KUKA KRL program: MyProgram_140().src

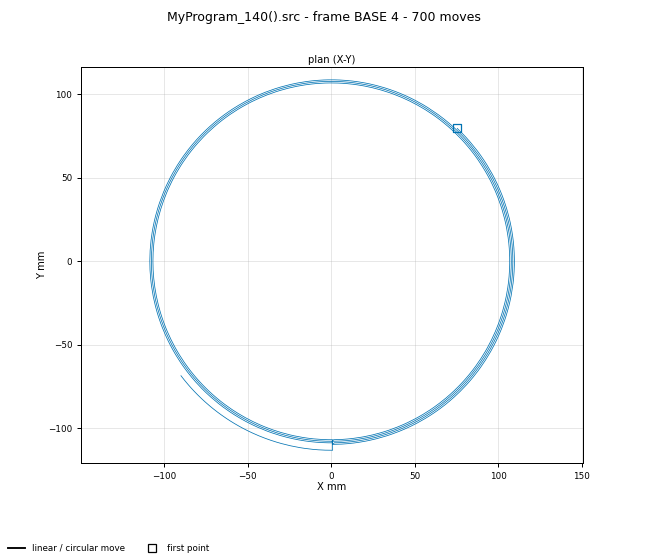
[picture p0: tool path of MyProgram_140().src in frame BASE 4, 700 of 700 moves have a stored position in this frame; points joined in program order, loops and branches not executed]
&ACCESS RVP
&REL 1
&PARAM TEMPLATE = C:\KRC\Roboter\Template\vorgabe
&PARAM EDITMASK = *
DEF MyProgram_140()
; ---- Setting reference (Base) ----
$BASE = BASE_DATA[4]

; --------------------------
; ---- Setting tool (TCP) ----
$TOOL = TOOL_DATA[3]
; --------------------------

$VEL.CP = VEL_APROX_PRINT
Startdeposition()
$VEL.CP = VEL_PRINT
LIN {X 75.377,Y 79.5533,Z 112,A 41.5429,B 24.9329,C -1.8914,E1 25.1111,E2 404.2043} C_DIS
LIN {X 77.9618,Y 77.0209,Z 112,A 39.7564,B 24.9329,C -1.8919,E1 25.1146,E2 405.9821} C_DIS
LIN {X 80.4801,Y 74.3866,Z 112,A 37.7745,B 24.9334,C -1.8843,E1 25.1184,E2 407.9731} C_DIS
LIN {X 82.9193,Y 71.6588,Z 112,A 35.8331,B 24.9338,C -1.8787,E1 25.122,E2 409.9192} C_DIS
LIN {X 87.2481,Y 66.3205,Z 112,A 32.4353,B 24.9338,C -1.8785,E1 25.1279,E2 413.3016} C_DIS
LIN {X 89.2094,Y 63.6549,Z 112,A 30.167,B 24.9358,C -1.8509,E1 25.1317,E2 415.624} C_DIS
LIN {X 91.3083,Y 60.6066,Z 112,A 28.6448,B 24.9349,C -1.8637,E1 25.134,E2 417.1083} C_DIS
LIN {X 93.1243,Y 57.7775,Z 112,A 27.0143,B 24.9349,C -1.8646,E1 25.1364,E2 418.7285} C_DIS
LIN {X 96.3793,Y 52.1661,Z 112,A 23.6682,B 24.9353,C -1.8574,E1 25.1411,E2 422.0744} C_DIS
LIN {X 97.758,Y 49.5356,Z 112,A 21.4703,B 24.9376,C -1.825,E1 25.1439,E2 424.3371} C_DIS
LIN {X 99.5673,Y 45.7914,Z 112,A 20.1073,B 24.9356,C -1.8541,E1 25.1455,E2 425.6239} C_DIS
LIN {X 101.01,Y 42.5115,Z 112,A 18.0918,B 24.9364,C -1.8425,E1 25.1477,E2 427.6559} C_DIS
LIN {X 102.2498,Y 39.4421,Z 112,A 15.9159,B 24.9381,C -1.8179,E1 25.15,E2 429.8778} C_DIS
LIN {X 103.3582,Y 36.433,Z 112,A 14.9671,B 24.9362,C -1.8448,E1 25.1508,E2 430.7576} C_DIS
LIN {X 104.9128,Y 31.6824,Z 112,A 11.8359,B 24.9383,C -1.8141,E1 25.1535,E2 433.9435} C_DIS
LIN {X 106.5712,Y 25.5542,Z 112,A 8.8976,B 24.9379,C -1.8206,E1 25.1556,E2 436.8496} C_DIS
LIN {X 107.1441,Y 23.0328,Z 112,A 7.4205,B 24.9385,C -1.8109,E1 25.1565,E2 438.341} C_DIS
LIN {X 107.8727,Y 19.3326,Z 112,A 5.4382,B 24.939,C -1.8042,E1 25.1575,E2 440.3275} C_DIS
LIN {X 108.4862,Y 15.5247,Z 112,A 3.44,B 24.9394,C -1.7986,E1 25.1583,E2 442.3271} C_DIS
LIN {X 108.9203,Y 12.1254,Z 112,A 1.543,B 24.9401,C -1.7882,E1 25.159,E2 444.2375} C_DIS
LIN {X 109.2712,Y 8.3779,Z 112,A -0.353,B 24.9403,C -1.7851,E1 25.1594,E2 446.1296} C_DIS
LIN {X 109.4863,Y 4.7961,Z 112,A -2.1281,B 24.9403,C -1.7835,E1 25.1597,E2 447.8979} C_DIS
LIN {X 109.5863,Y 1.1777,Z 112,A -4.0411,B 24.9409,C -1.7764,E1 25.1597,E2 449.8161} C_DIS
LIN {X 109.5675,Y -2.3032,Z 112,A -5.9034,B 24.9414,C -1.7686,E1 25.1597,E2 451.6858} C_DIS
LIN {X 109.4279,Y -5.9824,Z 112,A -7.7314,B 24.9415,C -1.7667,E1 25.1595,E2 453.5075} C_DIS
LIN {X 109.1646,Y -9.6696,Z 112,A -9.7033,B 24.942,C -1.7587,E1 25.159,E2 455.4866} C_DIS
LIN {X 108.816,Y -13.0152,Z 112,A -11.5187,B 24.9426,C -1.7504,E1 25.1585,E2 457.3107} C_DIS
LIN {X 107.6217,Y -20.684,Z 112,A -15.0658,B 24.9419,C -1.76,E1 25.1569,E2 460.8144} C_DIS
LIN {X 106.7931,Y -24.6068,Z 112,A -17.514,B 24.9434,C -1.7375,E1 25.1555,E2 463.3013} C_DIS
LIN {X 105.883,Y -28.2691,Z 112,A -19.5465,B 24.944,C -1.7286,E1 25.154,E2 465.3432} C_DIS
LIN {X 104.8011,Y -32.0495,Z 112,A -21.5394,B 24.9442,C -1.7248,E1 25.1525,E2 467.3336} C_DIS
LIN {X 103.8,Y -35.1546,Z 112,A -23.2039,B 24.9445,C -1.7213,E1 25.151,E2 468.9969} C_DIS
LIN {X 101.7907,Y -40.6108,Z 112,A -26.0892,B 24.9446,C -1.7186,E1 25.1482,E2 471.8725} C_DIS
LIN {X 100.2347,Y -44.3123,Z 112,A -28.8953,B 24.947,C -1.681,E1 25.145,E2 474.7519} C_DIS
LIN {X 98.5105,Y -48.0243,Z 112,A -30.3569,B 24.9456,C -1.7044,E1 25.1433,E2 476.1506} C_DIS
LIN {X 97.1937,Y -50.6336,Z 112,A -32.1386,B 24.9466,C -1.6886,E1 25.141,E2 477.96} C_DIS
LIN {X 95.3849,Y -53.9661,Z 112,A -34.0746,B 24.9468,C -1.6848,E1 25.1384,E2 479.8949} C_DIS
LIN {X 92.3521,Y -59.0034,Z 112,A -36.8045,B 24.9464,C -1.6912,E1 25.1345,E2 482.5959} C_DIS
LIN {X 89.3255,Y -63.492,Z 112,A -39.5066,B 24.9466,C -1.6888,E1 25.1303,E2 485.2901} C_DIS
LIN {X 87.7889,Y -65.6007,Z 112,A -41.8928,B 24.9496,C -1.6403,E1 25.1261,E2 487.7794} C_DIS
LIN {X 84.8508,Y -69.36,Z 112,A -44.0527,B 24.9491,C -1.6482,E1 25.1223,E2 489.9107} C_DIS
LIN {X 82.6946,Y -71.9159,Z 112,A -45.1241,B 24.9475,C -1.6733,E1 25.1205,E2 490.9181} C_DIS
LIN {X 80.8114,Y -74.0256,Z 112,A -46.889,B 24.9486,C -1.6569,E1 25.1171,E2 492.7137} C_DIS
LIN {X 77.0376,Y -77.9452,Z 112,A -50.0153,B 24.9498,C -1.6376,E1 25.1109,E2 495.8723} C_DIS
LIN {X 73.6027,Y -81.1994,Z 112,A -52.2586,B 24.9495,C -1.6417,E1 25.1064,E2 498.0968} C_DIS
LIN {X 70.6465,Y -83.7833,Z 112,A -54.5965,B 24.9505,C -1.6247,E1 25.1014,E2 500.4658} C_DIS
LIN {X 68.0835,Y -85.8773,Z 112,A -56.4348,B 24.9511,C -1.6162,E1 25.0973,E2 502.3171} C_DIS
LIN {X 64.9846,Y -88.246,Z 112,A -57.6863,B 24.9492,C -1.646,E1 25.0947,E2 503.4939} C_DIS
LIN {X 61.6206,Y -90.6267,Z 112,A -60.4571,B 24.9511,C -1.6149,E1 25.0882,E2 506.3286} C_DIS
LIN {X 58.8929,Y -92.423,Z 112,A -61.4446,B 24.9494,C -1.6427,E1 25.086,E2 507.2473} C_DIS
LIN {X 56.1138,Y -94.1364,Z 112,A -63.2822,B 24.95,C -1.6337,E1 25.0816,E2 509.1002} C_DIS
LIN {X 51.5128,Y -96.7304,Z 112,A -66.8077,B 24.9523,C -1.5961,E1 25.0728,E2 512.7044} C_DIS
LIN {X 47.8579,Y -98.5904,Z 112,A -68.1842,B 24.9505,C -1.6253,E1 25.0695,E2 514.0081} C_DIS
LIN {X 43.812,Y -100.4528,Z 112,A -70.6813,B 24.9512,C -1.6145,E1 25.0631,E2 516.5246} C_DIS
LIN {X 40.4857,Y -101.8399,Z 112,A -73.4033,B 24.9534,C -1.5763,E1 25.0559,E2 519.3307} C_DIS
LIN {X 35.6056,Y -103.6479,Z 112,A -75.1848,B 24.9513,C -1.6124,E1 25.0514,E2 521.0232} C_DIS
LIN {X 32.8161,Y -104.5634,Z 112,A -77.2633,B 24.9528,C -1.5876,E1 25.0457,E2 523.1566} C_DIS
LIN {X 29.377,Y -105.5818,Z 112,A -78.6243,B 24.9516,C -1.6072,E1 25.0422,E2 524.4689} C_DIS
LIN {X 27.077,Y -106.1938,Z 112,A -80.5198,B 24.9533,C -1.5786,E1 25.0369,E2 526.4294} C_DIS
LIN {X 23.0114,Y -107.1488,Z 112,A -81.9602,B 24.9516,C -1.6077,E1 25.0332,E2 527.7989} C_DIS
LIN {X 20.5758,Y -107.6425,Z 112,A -83.3737,B 24.9519,C -1.6018,E1 25.0292,E2 529.2248} C_DIS
LIN {X 16.5964,Y -108.3275,Z 112,A -85.5038,B 24.9521,C -1.5994,E1 25.0234,E2 531.3583} C_DIS
LIN {X 13.46,Y -108.7634,Z 112,A -87.2798,B 24.9524,C -1.5932,E1 25.0184,E2 533.1475} C_DIS
LIN {X 9.8662,Y -109.1465,Z 112,A -89.0287,B 24.9521,C -1.5981,E1 25.0136,E2 534.8837} C_DIS
LIN {X 6.2606,Y -109.4125,Z 112,A -90.9395,B 24.9522,C -1.5964,E1 25.0082,E2 536.7978} C_DIS
LIN {X 2.6896,Y -109.5604,Z 112,A -92.7328,B 24.9522,C -1.5988,E1 25.0033,E2 538.5848} C_DIS
LIN {X 0.7741,Y -109.5863,Z 112,A -93.6774,B 24.952,C -1.601,E1 25.0006,E2 539.5242} C_DIS
Enddeposition()
LIN {X 0.7741,Y -109.5863,Z 112,A -93.6774,B 24.952,C -1.601,E1 25.0006,E2 539.5242} C_DIS
Startdeposition()
$VEL.CP = VEL_PRINT
LIN {X 1.7946,Y -108.6458,Z 112,A -92.6033,B 24.9496,C -1.6396,E1 25.0039,E2 538.3587} C_DIS
LIN {X 4.823,Y -108.5535,Z 112,A -90.9393,B 24.9494,C -1.643,E1 25.0086,E2 536.6872} C_DIS
LIN {X 8.3887,Y -108.3365,Z 112,A -89.0175,B 24.9493,C -1.6454,E1 25.0139,E2 534.7604} C_DIS
LIN {X 11.9173,Y -108.0066,Z 112,A -87.0722,B 24.949,C -1.6497,E1 25.0193,E2 532.8063} C_DIS
LIN {X 15.0872,Y -107.6081,Z 112,A -85.4658,B 24.9491,C -1.6475,E1 25.0238,E2 531.2064} C_DIS
LIN {X 18.76,Y -107.0298,Z 112,A -83.4639,B 24.9489,C -1.6507,E1 25.0293,E2 529.1988} C_DIS
LIN {X 22.7045,Y -106.2629,Z 112,A -80.8395,B 24.9475,C -1.6741,E1 25.0366,E2 526.5224} C_DIS
LIN {X 26.6242,Y -105.349,Z 112,A -79.2573,B 24.9488,C -1.6532,E1 25.0408,E2 524.992} C_DIS
LIN {X 32.0291,Y -103.8328,Z 112,A -76.2746,B 24.9485,C -1.6575,E1 25.0488,E2 522.0042} C_DIS
LIN {X 35.4323,Y -102.7228,Z 112,A -74.419,B 24.9485,C -1.6585,E1 25.0537,E2 520.15} C_DIS
LIN {X 40.5582,Y -100.8083,Z 112,A -71.5163,B 24.9482,C -1.6632,E1 25.0613,E2 517.2424} C_DIS
LIN {X 43.2349,Y -99.6889,Z 112,A -69.482,B 24.9466,C -1.6873,E1 25.0666,E2 515.156} C_DIS
LIN {X 46.9131,Y -98.0116,Z 112,A -68.0486,B 24.9483,C -1.6605,E1 25.0701,E2 513.7897} C_DIS
LIN {X 48.9246,Y -97.0243,Z 112,A -66.0205,B 24.9459,C -1.6992,E1 25.0753,E2 511.6757} C_DIS
LIN {X 53.0461,Y -94.8325,Z 112,A -64.3618,B 24.9478,C -1.6686,E1 25.0792,E2 510.0941} C_DIS
LIN {X 56.0148,Y -93.1111,Z 112,A -62.5662,B 24.9477,C -1.6713,E1 25.0835,E2 508.2976} C_DIS
LIN {X 59.0835,Y -91.1945,Z 112,A -60.1603,B 24.9461,C -1.6967,E1 25.0893,E2 505.8395} C_DIS
LIN {X 61.9282,Y -89.2861,Z 112,A -58.7501,B 24.9469,C -1.6831,E1 25.0925,E2 504.4662} C_DIS
LIN {X 65.7981,Y -86.4746,Z 112,A -56.1025,B 24.9462,C -1.6939,E1 25.0984,E2 501.8027} C_DIS
LIN {X 70.9814,Y -82.2747,Z 112,A -52.6965,B 24.946,C -1.6968,E1 25.1057,E2 498.4027} C_DIS
LIN {X 73.5373,Y -79.996,Z 112,A -50.3929,B 24.9444,C -1.7231,E1 25.1106,E2 496.0464} C_DIS
LIN {X 76.5543,Y -77.1142,Z 112,A -48.1485,B 24.9439,C -1.7305,E1 25.115,E2 493.7941} C_DIS
LIN {X 79.6532,Y -73.911,Z 112,A -46.3962,B 24.9452,C -1.7099,E1 25.1183,E2 492.0981} C_DIS
LIN {X 81.5881,Y -71.7678,Z 112,A -44.2717,B 24.9432,C -1.7405,E1 25.1223,E2 489.9107} C_DIS
LIN {X 84.4673,Y -68.3547,Z 112,A -42.3211,B 24.944,C -1.7288,E1 25.1257,E2 487.9969} C_DIS
LIN {X 88.438,Y -63.1333,Z 112,A -38.1967,B 24.9414,C -1.7681,E1 25.1326,E2 483.7997} C_DIS
LIN {X 91.6609,Y -58.3569,Z 112,A -35.9253,B 24.9431,C -1.7424,E1 25.1359,E2 481.6004} C_DIS
LIN {X 93.7475,Y -54.9424,Z 112,A -34.0234,B 24.9433,C -1.7392,E1 25.1386,E2 479.7157} C_DIS
LIN {X 95.2658,Y -52.2666,Z 112,A -32.5867,B 24.9435,C -1.7358,E1 25.1406,E2 478.2946} C_DIS
LIN {X 97.5098,Y -47.9483,Z 112,A -29.1045,B 24.9403,C -1.7844,E1 25.1451,E2 474.7162} C_DIS
LIN {X 99.5831,Y -43.4777,Z 112,A -27.3196,B 24.9422,C -1.7559,E1 25.147,E2 473.0083} C_DIS
LIN {X 100.6196,Y -41.0219,Z 112,A -25.5416,B 24.9408,C -1.7769,E1 25.1489,E2 471.1906} C_DIS
LIN {X 101.8245,Y -37.9368,Z 112,A -24.2243,B 24.9417,C -1.7631,E1 25.1502,E2 469.9131} C_DIS
LIN {X 102.8382,Y -35.0935,Z 112,A -22.5787,B 24.9412,C -1.7705,E1 25.1517,E2 468.2593} C_DIS
LIN {X 103.8368,Y -32.0163,Z 112,A -20.9416,B 24.9411,C -1.7728,E1 25.1531,E2 466.626} C_DIS
LIN {X 104.7149,Y -29.0219,Z 112,A -19.1378,B 24.9403,C -1.7851,E1 25.1544,E2 464.8035} C_DIS
LIN {X 105.6382,Y -25.4512,Z 112,A -17.2444,B 24.94,C -1.7891,E1 25.1557,E2 462.9118} C_DIS
LIN {X 106.4295,Y -21.9056,Z 112,A -15.1285,B 24.939,C -1.8042,E1 25.157,E2 460.7725} C_DIS
LIN {X 107.4359,Y -16.2708,Z 112,A -12.2941,B 24.9389,C -1.8057,E1 25.1582,E2 457.9511} C_DIS
LIN {X 107.9465,Y -12.4376,Z 112,A -10.3554,B 24.9387,C -1.8079,E1 25.1589,E2 456.0188} C_DIS
LIN {X 108.3235,Y -8.5506,Z 112,A -8.3385,B 24.9384,C -1.8127,E1 25.1594,E2 454.0025} C_DIS
LIN {X 108.5553,Y -4.7801,Z 112,A -6.3472,B 24.938,C -1.8191,E1 25.1597,E2 452.0079} C_DIS
LIN {X 108.6585,Y -0.7391,Z 112,A -4.2535,B 24.9376,C -1.8244,E1 25.1597,E2 449.9143} C_DIS
LIN {X 108.6205,Y 2.9676,Z 112,A -2.291,B 24.9372,C -1.831,E1 25.1597,E2 447.9477} C_DIS
LIN {X 108.4705,Y 6.4379,Z 112,A -0.4958,B 24.9369,C -1.8353,E1 25.1594,E2 446.1531} C_DIS
LIN {X 108.2062,Y 9.925,Z 112,A 1.3366,B 24.9365,C -1.8408,E1 25.159,E2 444.3188} C_DIS
LIN {X 107.7971,Y 13.6733,Z 112,A 3.2648,B 24.9362,C -1.8444,E1 25.1584,E2 442.3932} C_DIS
LIN {X 107.4067,Y 16.4592,Z 112,A 4.7603,B 24.9359,C -1.8497,E1 25.1578,E2 440.8942} C_DIS
LIN {X 106.8273,Y 19.8864,Z 112,A 6.707,B 24.9351,C -1.8605,E1 25.1568,E2 438.9333} C_DIS
LIN {X 106.1072,Y 23.4184,Z 112,A 8.4034,B 24.9353,C -1.8574,E1 25.1558,E2 437.2542} C_DIS
LIN {X 104.6842,Y 29.1302,Z 112,A 12.1394,B 24.9327,C -1.8951,E1 25.1531,E2 433.4508} C_DIS
LIN {X 103.5197,Y 33.0295,Z 112,A 13.8129,B 24.9337,C -1.8806,E1 25.1518,E2 431.821} C_DIS
LIN {X 102.3599,Y 36.4666,Z 112,A 15.4437,B 24.9342,C -1.8738,E1 25.1503,E2 430.2153} C_DIS
LIN {X 101.3028,Y 39.307,Z 112,A 17.1938,B 24.9334,C -1.8853,E1 25.1485,E2 428.448} C_DIS
LIN {X 100.0814,Y 42.3182,Z 112,A 18.9048,B 24.933,C -1.8902,E1 25.1467,E2 426.7348} C_DIS
LIN {X 98.6024,Y 45.6585,Z 112,A 21.3213,B 24.9311,C -1.9174,E1 25.1438,E2 424.2673} C_DIS
LIN {X 96.9145,Y 49.1405,Z 112,A 22.8666,B 24.9322,C -1.9012,E1 25.142,E2 422.7683} C_DIS
LIN {X 95.2954,Y 52.212,Z 112,A 25.2882,B 24.93,C -1.9323,E1 25.1386,E2 420.286} C_DIS
LIN {X 93.1242,Y 55.9932,Z 112,A 27.0114,B 24.9314,C -1.9131,E1 25.1363,E2 418.6171} C_DIS
LIN {X 91.2048,Y 59.0675,Z 112,A 28.8675,B 24.9312,C -1.9157,E1 25.1335,E2 416.7641} C_DIS
LIN {X 87.762,Y 64.0698,Z 112,A 31.9965,B 24.9308,C -1.9206,E1 25.1285,E2 413.6389} C_DIS
LIN {X 83.1642,Y 69.9372,Z 112,A 36.026,B 24.9299,C -1.9342,E1 25.1214,E2 409.5959} C_DIS
LIN {X 80.7592,Y 72.6989,Z 112,A 37.9225,B 24.9296,C -1.9372,E1 25.1179,E2 407.701} C_DIS
LIN {X 78.2275,Y 75.4158,Z 112,A 39.7969,B 24.9296,C -1.9379,E1 25.1143,E2 405.833} C_DIS
LIN {X 75.5755,Y 78.0736,Z 112,A 41.7857,B 24.9293,C -1.9425,E1 25.1104,E2 403.8417} C_DIS
LIN {X 72.9803,Y 80.5071,Z 112,A 43.7462,B 24.9287,C -1.95,E1 25.1063,E2 401.8715} C_DIS
LIN {X 70.3797,Y 82.7877,Z 112,A 45.4481,B 24.9288,C -1.9483,E1 25.1027,E2 400.1801} C_DIS
LIN {X 67.5295,Y 85.1287,Z 112,A 48.0314,B 24.9265,C -1.9795,E1 25.097,E2 397.5329} C_DIS
LIN {X 64.0831,Y 87.7523,Z 112,A 49.6382,B 24.9284,C -1.9544,E1 25.0935,E2 395.9912} C_DIS
LIN {X 57.7373,Y 92.0518,Z 112,A 53.6998,B 24.9278,C -1.9617,E1 25.0841,E2 391.9257} C_DIS
LIN {X 54.769,Y 93.8499,Z 112,A 55.4275,B 24.928,C -1.9601,E1 25.0799,E2 390.2073} C_DIS
LIN {X 49.9797,Y 96.4856,Z 112,A 58.3902,B 24.9274,C -1.9674,E1 25.0726,E2 387.2358} C_DIS
LIN {X 47.5326,Y 97.714,Z 112,A 60.3077,B 24.9258,C -1.9892,E1 25.0677,E2 385.2717} C_DIS
LIN {X 44.2589,Y 99.2392,Z 112,A 61.825,B 24.9269,C -1.9751,E1 25.0639,E2 383.7917} C_DIS
LIN {X 40.9639,Y 100.6432,Z 112,A 63.5708,B 24.9272,C -1.9711,E1 25.0595,E2 382.0593} C_DIS
LIN {X 38.3632,Y 101.663,Z 112,A 65.5197,B 24.9256,C -1.9925,E1 25.0543,E2 380.064} C_DIS
LIN {X 35.071,Y 102.8458,Z 112,A 66.9096,B 24.9269,C -1.975,E1 25.0507,E2 378.7182} C_DIS
LIN {X 31.9792,Y 103.8483,Z 112,A 68.6432,B 24.9267,C -1.9772,E1 25.0461,E2 376.9826} C_DIS
LIN {X 27.1829,Y 105.2055,Z 112,A 71.8741,B 24.9247,C -2.004,E1 25.0372,E2 373.6933} C_DIS
LIN {X 23.0994,Y 106.1768,Z 112,A 73.4715,B 24.9265,C -1.9796,E1 25.033,E2 372.156} C_DIS
LIN {X 20.474,Y 106.7142,Z 112,A 74.9013,B 24.9265,C -1.9809,E1 25.0291,E2 370.7248} C_DIS
LIN {X 16.3963,Y 107.4165,Z 112,A 77.1625,B 24.9261,C -1.9848,E1 25.0228,E2 368.4565} C_DIS
LIN {X 12.6448,Y 107.9222,Z 112,A 79.0915,B 24.9263,C -1.9825,E1 25.0175,E2 366.5344} C_DIS
LIN {X 8.7801,Y 108.3052,Z 112,A 81.1507,B 24.9263,C -1.9832,E1 25.0118,E2 364.4749} C_DIS
LIN {X 5.1053,Y 108.5413,Z 112,A 83.076,B 24.9263,C -1.9825,E1 25.0064,E2 362.552} C_DIS
LIN {X 2.0105,Y 108.6418,Z 112,A 84.7124,B 24.9263,C -1.9825,E1 25.0019,E2 360.916} C_DIS
LIN {X -1.8793,Y 108.6443,Z 112,A 86.6636,B 24.9266,C -1.9779,E1 24.9964,E2 358.9755} C_DIS
LIN {X -4.5203,Y 108.5665,Z 112,A 88.1228,B 24.9265,C -1.9802,E1 24.9924,E2 357.5107} C_DIS
LIN {X -8.1438,Y 108.3561,Z 112,A 90.1157,B 24.9263,C -1.9825,E1 24.9868,E2 355.5114} C_DIS
LIN {X -11.5164,Y 108.0486,Z 112,A 91.9035,B 24.9263,C -1.9817,E1 24.9818,E2 353.7246} C_DIS
LIN {X -15.1504,Y 107.5991,Z 112,A 93.6701,B 24.9269,C -1.974,E1 24.977,E2 351.9751} C_DIS
LIN {X -20.548,Y 106.6999,Z 112,A 97.2399,B 24.9251,C -1.9992,E1 24.967,E2 348.3418} C_DIS
LIN {X -24.5356,Y 105.8542,Z 112,A 98.7968,B 24.927,C -1.9735,E1 24.9629,E2 346.8438} C_DIS
LIN {X -30.2104,Y 104.3781,Z 112,A 102.4845,B 24.9255,C -1.994,E1 24.9528,E2 343.1018} C_DIS
LIN {X -34.0854,Y 103.1781,Z 112,A 104.1442,B 24.9271,C -1.9724,E1 24.9486,E2 341.4904} C_DIS
LIN {X -37.0469,Y 102.1502,Z 112,A 105.7169,B 24.9274,C -1.9672,E1 24.9444,E2 339.927} C_DIS
LIN {X -39.4458,Y 101.2483,Z 112,A 107.5174,B 24.9263,C -1.983,E1 24.9397,E2 338.0849} C_DIS
LIN {X -42.7406,Y 99.9027,Z 112,A 109.0294,B 24.9275,C -1.9659,E1 24.9359,E2 336.61} C_DIS
LIN {X -45.2802,Y 98.7785,Z 112,A 110.8572,B 24.9266,C -1.978,E1 24.9312,E2 334.7491} C_DIS
LIN {X -48.3038,Y 97.3336,Z 112,A 112.6602,B 24.9268,C -1.9765,E1 24.9266,E2 332.9447} C_DIS
LIN {X -51.5219,Y 95.6697,Z 112,A 114.406,B 24.9275,C -1.9668,E1 24.9224,E2 331.2171} C_DIS
LIN {X -55.5157,Y 93.4086,Z 112,A 116.6397,B 24.9283,C -1.9552,E1 24.917,E2 329.0044} C_DIS
LIN {X -59.0398,Y 91.2226,Z 112,A 118.6379,B 24.9292,C -1.9438,E1 24.9124,E2 327.0271} C_DIS
LIN {X -61.302,Y 89.7182,Z 112,A 120.6482,B 24.9277,C -1.9633,E1 24.9076,E2 324.9635} C_DIS
LIN {X -64.2075,Y 87.6612,Z 112,A 122.0568,B 24.9293,C -1.9413,E1 24.9045,E2 323.6024} C_DIS
LIN {X -67.0333,Y 85.5209,Z 112,A 123.7482,B 24.9301,C -1.9305,E1 24.9008,E2 321.9306} C_DIS
LIN {X -69.5994,Y 83.4449,Z 112,A 126.1945,B 24.9284,C -1.9538,E1 24.8954,E2 319.4194} C_DIS
LIN {X -72.4368,Y 80.9939,Z 112,A 127.6579,B 24.9302,C -1.9295,E1 24.8925,E2 318.0081} C_DIS
LIN {X -75.1131,Y 78.5193,Z 112,A 129.4026,B 24.931,C -1.9182,E1 24.889,E2 316.2833} C_DIS
LIN {X -78.1859,Y 75.459,Z 112,A 132.3647,B 24.9296,C -1.9384,E1 24.883,E2 313.2602} C_DIS
LIN {X -80.6542,Y 72.8162,Z 112,A 133.8743,B 24.931,C -1.9184,E1 24.8803,E2 311.7917} C_DIS
LIN {X -83.1284,Y 69.9798,Z 112,A 135.722,B 24.9318,C -1.908,E1 24.8769,E2 309.9603} C_DIS
LIN {X -85.5795,Y 66.9591,Z 112,A 138.1312,B 24.9312,C -1.9162,E1 24.8727,E2 307.5203} C_DIS
LIN {X -88.378,Y 63.2174,Z 112,A 140.3479,B 24.9323,C -1.9001,E1 24.8691,E2 305.3313} C_DIS
LIN {X -90.2079,Y 60.5789,Z 112,A 142.5634,B 24.9312,C -1.9152,E1 24.8656,E2 303.0687} C_DIS
LIN {X -92.2077,Y 57.4877,Z 112,A 144.9067,B 24.9305,C -1.9251,E1 24.8621,E2 300.69} C_DIS
LIN {X -94.9198,Y 52.8897,Z 112,A 146.7523,B 24.9337,C -1.88,E1 24.8597,E2 298.9423} C_DIS
LIN {X -96.5074,Y 49.937,Z 112,A 148.4926,B 24.9342,C -1.8737,E1 24.8574,E2 297.2076} C_DIS
LIN {X -98.8674,Y 45.0839,Z 112,A 151.562,B 24.9342,C -1.8735,E1 24.8537,E2 294.122} C_DIS
LIN {X -100.4255,Y 41.4987,Z 112,A 153.677,B 24.9345,C -1.8692,E1 24.8514,E2 292.0055} C_DIS
LIN {X -102.9015,Y 34.9056,Z 112,A 157.3268,B 24.9355,C -1.8553,E1 24.8479,E2 288.3684} C_DIS
LIN {X -103.9854,Y 31.5367,Z 112,A 159.105,B 24.9361,C -1.8461,E1 24.8464,E2 286.6019} C_DIS
LIN {X -105.2366,Y 27.0621,Z 112,A 161.5783,B 24.9366,C -1.8391,E1 24.8446,E2 284.1308} C_DIS
LIN {X -105.9082,Y 24.3015,Z 112,A 163.0977,B 24.9369,C -1.8352,E1 24.8436,E2 282.612} C_DIS
LIN {X -106.6422,Y 20.8479,Z 112,A 165.0036,B 24.9372,C -1.8308,E1 24.8426,E2 280.7052} C_DIS
LIN {X -107.2342,Y 17.5517,Z 112,A 167.1449,B 24.9366,C -1.8392,E1 24.8415,E2 278.531} C_DIS
LIN {X -107.9134,Y 12.7198,Z 112,A 170.4744,B 24.9352,C -1.8596,E1 24.8404,E2 275.1329} C_DIS
LIN {X -108.4608,Y 6.6128,Z 112,A 173.8021,B 24.9357,C -1.8527,E1 24.8399,E2 271.8017} C_DIS
LIN {X -108.6618,Y 0.2533,Z 112,A 176.387,B 24.9384,C -1.8125,E1 24.8399,E2 269.2972} C_DIS
LIN {X -108.54,Y -5.1359,Z 112,A 179.8158,B 24.9375,C -1.8256,E1 24.8402,E2 265.8164} C_DIS
LIN {X -108.1471,Y -10.5661,Z 112,A -178.3924,B 24.9409,C -1.7755,E1 24.8406,E2 264.1334} C_DIS
LIN {X -107.6869,Y -14.5242,Z 112,A -175.976,B 24.9406,C -1.7807,E1 24.8415,E2 261.6903} C_DIS
LIN {X -106.5874,Y -21.1321,Z 112,A -172.4385,B 24.9413,C -1.7697,E1 24.8432,E2 258.158} C_DIS
LIN {X -105.2808,Y -26.89,Z 112,A -169.3783,B 24.9421,C -1.758,E1 24.8451,E2 255.1076} C_DIS
LIN {X -104.2561,Y -30.6242,Z 112,A -167.3737,B 24.9426,C -1.7504,E1 24.8466,E2 253.1096} C_DIS
LIN {X -103.3385,Y -33.5896,Z 112,A -165.6133,B 24.9426,C -1.7501,E1 24.8481,E2 251.3398} C_DIS
LIN {X -102.0931,Y -37.2033,Z 112,A -163.6489,B 24.9431,C -1.7422,E1 24.85,E2 249.3832} C_DIS
LIN {X -101.1257,Y -39.7577,Z 112,A -161.6196,B 24.9419,C -1.7605,E1 24.8521,E2 247.2989} C_DIS
LIN {X -99.5429,Y -43.5699,Z 112,A -159.4525,B 24.9424,C -1.7538,E1 24.8545,E2 245.1358} C_DIS
LIN {X -97.8597,Y -47.2292,Z 112,A -157.9217,B 24.9442,C -1.7251,E1 24.8563,E2 243.6651} C_DIS
LIN {X -96.3833,Y -50.1758,Z 112,A -156.1673,B 24.9445,C -1.7209,E1 24.8585,E2 241.9114} C_DIS
LIN {X -94.8115,Y -53.0837,Z 112,A -154.3953,B 24.9447,C -1.7172,E1 24.8609,E2 240.1388} C_DIS
LIN {X -93.0799,Y -56.066,Z 112,A -152.7498,B 24.9455,C -1.7057,E1 24.8632,E2 238.5121} C_DIS
LIN {X -90.4621,Y -60.1989,Z 112,A -149.9648,B 24.9455,C -1.7068,E1 24.8675,E2 235.7104} C_DIS
LIN {X -88.4639,Y -63.097,Z 112,A -148.1296,B 24.9458,C -1.7014,E1 24.8704,E2 233.8792} C_DIS
LIN {X -86.322,Y -65.9983,Z 112,A -145.9458,B 24.9454,C -1.7076,E1 24.8741,E2 231.6702} C_DIS
LIN {X -83.6193,Y -69.3896,Z 112,A -143.9562,B 24.9464,C -1.6907,E1 24.8775,E2 229.7116} C_DIS
LIN {X -81.0033,Y -72.4262,Z 112,A -141.4118,B 24.9457,C -1.7026,E1 24.8823,E2 227.1273} C_DIS
LIN {X -77.4898,Y -76.1741,Z 112,A -139.053,B 24.9469,C -1.683,E1 24.8868,E2 224.8049} C_DIS
LIN {X -75.046,Y -78.5839,Z 112,A -137.1516,B 24.9469,C -1.6828,E1 24.8906,E2 222.8962} C_DIS
LIN {X -72.4875,Y -80.9485,Z 112,A -135.4484,B 24.9475,C -1.6739,E1 24.8941,E2 221.2073} C_DIS
LIN {X -67.8174,Y -84.9012,Z 112,A -132.0577,B 24.9475,C -1.6741,E1 24.9014,E2 217.8031} C_DIS
LIN {X -64.9179,Y -87.1375,Z 112,A -130.3708,B 24.9483,C -1.6611,E1 24.9051,E2 216.141} C_DIS
LIN {X -60.8905,Y -89.9969,Z 112,A -127.6157,B 24.9482,C -1.6627,E1 24.9115,E2 213.3728} C_DIS
LIN {X -57.7878,Y -92.0203,Z 112,A -125.8994,B 24.949,C -1.6502,E1 24.9154,E2 211.6805} C_DIS
LIN {X -53.5907,Y -94.5274,Z 112,A -122.9887,B 24.9484,C -1.6596,E1 24.9225,E2 208.7386} C_DIS
LIN {X -50.5833,Y -96.1687,Z 112,A -121.4619,B 24.9492,C -1.6461,E1 24.9262,E2 207.2397} C_DIS
LIN {X -47.2013,Y -97.8731,Z 112,A -119.2543,B 24.9489,C -1.652,E1 24.9317,E2 205.0122} C_DIS
LIN {X -43.9959,Y -99.3572,Z 112,A -117.2434,B 24.9486,C -1.6559,E1 24.9369,E2 202.9873} C_DIS
LIN {X -38.4006,Y -101.6489,Z 112,A -114.2252,B 24.9492,C -1.6459,E1 24.9447,E2 199.9862} C_DIS
LIN {X -35.6434,Y -102.6487,Z 112,A -112.4998,B 24.9489,C -1.6517,E1 24.9493,E2 198.2435} C_DIS
LIN {X -30.4712,Y -104.3015,Z 112,A -109.1993,B 24.9479,C -1.6675,E1 24.9582,E2 194.8999} C_DIS
LIN {X -26.7056,Y -105.3282,Z 112,A -107.5898,B 24.9491,C -1.6479,E1 24.9624,E2 193.3345} C_DIS
LIN {X -23.1015,Y -106.1763,Z 112,A -105.6893,B 24.9493,C -1.6449,E1 24.9676,E2 191.4388} C_DIS
LIN {X -19.429,Y -106.9095,Z 112,A -103.7369,B 24.9494,C -1.6432,E1 24.9729,E2 189.4883} C_DIS
LIN {X -15.8278,Y -107.5029,Z 112,A -101.7903,B 24.9494,C -1.6436,E1 24.9783,E2 187.5391} C_DIS
LIN {X -12.5986,Y -107.9276,Z 112,A -100.1107,B 24.9494,C -1.6418,E1 24.983,E2 185.8627} C_DIS
LIN {X -9.0922,Y -108.2802,Z 112,A -98.2047,B 24.9494,C -1.6436,E1 24.9883,E2 183.9513} C_DIS
LIN {X -5.4936,Y -108.5227,Z 112,A -96.2484,B 24.9492,C -1.6459,E1 24.9938,E2 181.9889} C_DIS
LIN {X -1.8138,Y -108.6455,Z 112,A -94.3542,B 24.9493,C -1.6443,E1 24.999,E2 180.0984} C_DIS
LIN {X 0.7652,Y -108.6557,Z 112,A -93.3115,B 24.9501,C -1.6315,E1 25.0019,E2 179.0861} C_DIS
Enddeposition()
LIN {X 0.7652,Y -108.6557,Z 112,A -93.3115,B 24.9501,C -1.6315,E1 25.0019,E2 179.0861} C_DIS
Startdeposition()
$VEL.CP = VEL_PRINT
LIN {X 0.2756,Y -107.7299,Z 112,A -94.2394,B 24.9508,C -1.6203,E1 24.9992,E2 180.0403} C_DIS
LIN {X -3.43,Y -107.675,Z 112,A -96.0829,B 24.9505,C -1.6252,E1 24.9941,E2 181.8725} C_DIS
LIN {X -7.1756,Y -107.4904,Z 112,A -98.1361,B 24.9507,C -1.6227,E1 24.9883,E2 183.9322} C_DIS
LIN {X -10.3726,Y -107.2301,Z 112,A -99.9153,B 24.9508,C -1.6199,E1 24.9834,E2 185.719} C_DIS
LIN {X -13.9001,Y -106.8291,Z 112,A -101.7029,B 24.9506,C -1.6242,E1 24.9784,E2 187.4976} C_DIS
LIN {X -17.8057,Y -106.2479,Z 112,A -103.8279,B 24.9506,C -1.6238,E1 24.9726,E2 189.6254} C_DIS
LIN {X -20.7424,Y -105.7145,Z 112,A -105.2905,B 24.9503,C -1.6294,E1 24.9686,E2 191.0764} C_DIS
LIN {X -23.2491,Y -105.1914,Z 112,A -106.85,B 24.9507,C -1.6221,E1 24.9643,E2 192.655} C_DIS
LIN {X -27.6838,Y -104.1127,Z 112,A -108.9884,B 24.9499,C -1.635,E1 24.9586,E2 194.7659} C_DIS
LIN {X -32.2563,Y -102.7878,Z 112,A -111.6063,B 24.95,C -1.6333,E1 24.9515,E2 197.3921} C_DIS
LIN {X -35.1519,Y -101.8347,Z 112,A -113.2079,B 24.9499,C -1.6354,E1 24.9473,E2 198.9918} C_DIS
LIN {X -37.145,Y -101.1235,Z 112,A -114.5386,B 24.9503,C -1.6283,E1 24.9437,E2 200.3419} C_DIS
LIN {X -40.6983,Y -99.7463,Z 112,A -116.2804,B 24.9495,C -1.6415,E1 24.9393,E2 202.0562} C_DIS
LIN {X -43.0152,Y -98.7692,Z 112,A -117.87,B 24.95,C -1.6331,E1 24.9352,E2 203.6696} C_DIS
LIN {X -46.0406,Y -97.3978,Z 112,A -119.7868,B 24.9503,C -1.6292,E1 24.9303,E2 205.6002} C_DIS
LIN {X -49.3103,Y -95.7823,Z 112,A -121.5156,B 24.9496,C -1.6399,E1 24.926,E2 207.3084} C_DIS
LIN {X -52.6225,Y -94.0029,Z 112,A -123.5606,B 24.9496,C -1.6408,E1 24.921,E2 209.3569} C_DIS
LIN {X -55.9844,Y -92.0403,Z 112,A -125.4675,B 24.949,C -1.6502,E1 24.9164,E2 211.2474} C_DIS
LIN {X -58.2159,Y -90.6453,Z 112,A -127.0417,B 24.9493,C -1.6456,E1 24.9127,E2 212.8375} C_DIS
LIN {X -61.8816,Y -88.1848,Z 112,A -129.3772,B 24.949,C -1.6499,E1 24.9073,E2 215.1706} C_DIS
LIN {X -64.6018,Y -86.2107,Z 112,A -131.199,B 24.9489,C -1.6517,E1 24.9032,E2 216.9945} C_DIS
LIN {X -67.2991,Y -84.1243,Z 112,A -133.3216,B 24.9494,C -1.6432,E1 24.8985,E2 219.1453} C_DIS
LIN {X -71.2456,Y -80.8083,Z 112,A -135.6521,B 24.9481,C -1.6642,E1 24.8936,E2 221.4349} C_DIS
LIN {X -73.2211,Y -79.0228,Z 112,A -137.1973,B 24.9482,C -1.6621,E1 24.8904,E2 222.9912} C_DIS
LIN {X -75.654,Y -76.6951,Z 112,A -139.0467,B 24.9482,C -1.6637,E1 24.8867,E2 224.8447} C_DIS
LIN {X -78.4163,Y -73.8685,Z 112,A -142.1078,B 24.9501,C -1.6324,E1 24.8807,E2 227.9936} C_DIS
LIN {X -82.2721,Y -69.5495,Z 112,A -144.0639,B 24.947,C -1.6814,E1 24.8773,E2 229.8418} C_DIS
LIN {X -84.0406,Y -67.4024,Z 112,A -145.6106,B 24.947,C -1.6824,E1 24.8746,E2 231.3933} C_DIS
LIN {X -85.7901,Y -65.1618,Z 112,A -147.3012,B 24.9472,C -1.6793,E1 24.8717,E2 233.0993} C_DIS
LIN {X -88.0351,Y -62.0952,Z 112,A -149.1436,B 24.9464,C -1.6911,E1 24.8687,E2 234.9226} C_DIS
LIN {X -89.7047,Y -59.6567,Z 112,A -150.8366,B 24.9464,C -1.6906,E1 24.866,E2 236.6253} C_DIS
LIN {X -91.7764,Y -56.4186,Z 112,A -152.7391,B 24.9458,C -1.7012,E1 24.8632,E2 238.5121} C_DIS
LIN {X -93.497,Y -53.5165,Z 112,A -154.6665,B 24.9458,C -1.7012,E1 24.8605,E2 240.4497} C_DIS
LIN {X -95.2879,Y -50.2582,Z 112,A -156.7483,B 24.9457,C -1.7027,E1 24.8577,E2 242.5388} C_DIS
LIN {X -97.0115,Y -46.8452,Z 112,A -158.9091,B 24.9457,C -1.7037,E1 24.855,E2 244.7089} C_DIS
LIN {X -98.6182,Y -43.3616,Z 112,A -160.8628,B 24.945,C -1.7127,E1 24.8528,E2 246.6518} C_DIS
LIN {X -100.3844,Y -39.0989,Z 112,A -163.2604,B 24.9444,C -1.7219,E1 24.8503,E2 249.0407} C_DIS
LIN {X -101.6417,Y -35.702,Z 112,A -165.2249,B 24.9442,C -1.7263,E1 24.8484,E2 251.006} C_DIS
LIN {X -102.6381,Y -32.7306,Z 112,A -166.7438,B 24.9435,C -1.7367,E1 24.8471,E2 252.5087} C_DIS
LIN {X -103.5372,Y -29.7636,Z 112,A -168.564,B 24.9435,C -1.7354,E1 24.8457,E2 254.3425} C_DIS
LIN {X -104.4289,Y -26.4648,Z 112,A -170.4525,B 24.9434,C -1.7384,E1 24.8444,E2 256.2349} C_DIS
LIN {X -105.1102,Y -23.6204,Z 112,A -171.9582,B 24.9429,C -1.745,E1 24.8434,E2 257.7336} C_DIS
LIN {X -105.7908,Y -20.3462,Z 112,A -173.8806,B 24.9429,C -1.7454,E1 24.8424,E2 259.6666} C_DIS
LIN {X -106.8035,Y -14.0976,Z 112,A -176.813,B 24.9412,C -1.772,E1 24.8411,E2 262.5531} C_DIS
LIN {X -107.2577,Y -10.0734,Z 112,A -179.6329,B 24.9423,C -1.7545,E1 24.8403,E2 265.4315} C_DIS
LIN {X -107.5109,Y -6.8712,Z 112,A 178.7333,B 24.9418,C -1.7627,E1 24.84,E2 267.0556} C_DIS
LIN {X -107.7035,Y -2.4083,Z 112,A 176.5706,B 24.9407,C -1.7781,E1 24.8398,E2 269.1945} C_DIS
LIN {X -107.7245,Y 1.1862,Z 112,A 174.1367,B 24.9416,C -1.7654,E1 24.8398,E2 271.6736} C_DIS
LIN {X -107.6087,Y 5.1272,Z 112,A 172.8235,B 24.9392,C -1.8006,E1 24.84,E2 272.9105} C_DIS
LIN {X -107.1606,Y 11.0583,Z 112,A 169.6467,B 24.9386,C -1.8104,E1 24.8407,E2 276.0831} C_DIS
LIN {X -106.8455,Y 13.7733,Z 112,A 167.6518,B 24.9396,C -1.7954,E1 24.8414,E2 278.1257} C_DIS
LIN {X -106.2943,Y 17.528,Z 112,A 165.8411,B 24.9386,C -1.8094,E1 24.8422,E2 279.9137} C_DIS
LIN {X -105.5575,Y 21.5241,Z 112,A 163.6814,B 24.9382,C -1.8164,E1 24.8433,E2 282.0695} C_DIS
LIN {X -104.6846,Y 25.4325,Z 112,A 161.5376,B 24.9377,C -1.8227,E1 24.8447,E2 284.2108} C_DIS
LIN {X -103.9361,Y 28.3375,Z 112,A 159.8425,B 24.9377,C -1.8242,E1 24.8459,E2 285.9123} C_DIS
LIN {X -103.1064,Y 31.2266,Z 112,A 158.4528,B 24.9368,C -1.8368,E1 24.847,E2 287.28} C_DIS
LIN {X -102.3156,Y 33.7273,Z 112,A 156.6257,B 24.9375,C -1.8255,E1 24.8486,E2 289.1446} C_DIS
LIN {X -101.0819,Y 37.2591,Z 112,A 154.9429,B 24.9363,C -1.8428,E1 24.8502,E2 290.7955} C_DIS
LIN {X -99.811,Y 40.5393,Z 112,A 153.0596,B 24.936,C -1.8482,E1 24.8521,E2 292.6766} C_DIS
LIN {X -98.3596,Y 43.945,Z 112,A 151.0641,B 24.9356,C -1.8532,E1 24.8543,E2 294.6712} C_DIS
LIN {X -96.9479,Y 46.9776,Z 112,A 149.1036,B 24.9357,C -1.8519,E1 24.8567,E2 296.6454} C_DIS
LIN {X -95.372,Y 50.0984,Z 112,A 147.3905,B 24.935,C -1.8628,E1 24.8589,E2 298.3417} C_DIS
LIN {X -92.8705,Y 54.5966,Z 112,A 144.6245,B 24.9345,C -1.8697,E1 24.8627,E2 301.1056} C_DIS
LIN {X -90.95,Y 57.7413,Z 112,A 142.5891,B 24.9343,C -1.8725,E1 24.8657,E2 303.1448} C_DIS
LIN {X -88.6858,Y 61.1609,Z 112,A 140.6803,B 24.9331,C -1.8886,E1 24.8686,E2 305.0245} C_DIS
LIN {X -86.8477,Y 63.7429,Z 112,A 138.8596,B 24.9331,C -1.8883,E1 24.8716,E2 306.855} C_DIS
LIN {X -84.9014,Y 66.3158,Z 112,A 136.9422,B 24.9334,C -1.8854,E1 24.8749,E2 308.7883} C_DIS
LIN {X -82.6529,Y 69.096,Z 112,A 135.1335,B 24.9328,C -1.8939,E1 24.8781,E2 310.5853} C_DIS
LIN {X -80.2042,Y 71.9232,Z 112,A 133.1873,B 24.9323,C -1.9006,E1 24.8816,E2 312.5243} C_DIS
LIN {X -77.7823,Y 74.5364,Z 112,A 131.2131,B 24.9322,C -1.9023,E1 24.8854,E2 314.5029} C_DIS
LIN {X -75.553,Y 76.7948,Z 112,A 129.6463,B 24.9315,C -1.9109,E1 24.8885,E2 316.0558} C_DIS
LIN {X -73.5696,Y 78.6974,Z 112,A 128.0778,B 24.9315,C -1.9104,E1 24.8917,E2 317.632} C_DIS
LIN {X -70.882,Y 81.1258,Z 112,A 126.0448,B 24.9315,C -1.9109,E1 24.896,E2 319.672} C_DIS
LIN {X -68.144,Y 83.4399,Z 112,A 124.4596,B 24.9304,C -1.9271,E1 24.8993,E2 321.2245} C_DIS
LIN {X -65.8287,Y 85.2775,Z 112,A 122.6306,B 24.9308,C -1.9209,E1 24.9034,E2 323.0752} C_DIS
LIN {X -63.4231,Y 87.0819,Z 112,A 120.2711,B 24.9326,C -1.8959,E1 24.9089,E2 325.5024} C_DIS
LIN {X -59.4002,Y 89.8738,Z 112,A 118.2095,B 24.9308,C -1.9212,E1 24.9135,E2 327.5106} C_DIS
LIN {X -56.492,Y 91.7317,Z 112,A 116.7018,B 24.9297,C -1.9369,E1 24.917,E2 328.9856} C_DIS
LIN {X -54.6875,Y 92.8168,Z 112,A 115.5152,B 24.9297,C -1.9365,E1 24.9199,E2 330.1769} C_DIS
LIN {X -51.441,Y 94.6546,Z 112,A 112.6462,B 24.9318,C -1.9067,E1 24.9271,E2 333.125} C_DIS
LIN {X -46.8795,Y 96.995,Z 112,A 111.038,B 24.9285,C -1.9533,E1 24.9308,E2 334.6265} C_DIS
LIN {X -43.0498,Y 98.7541,Z 112,A 108.1472,B 24.93,C -1.9319,E1 24.9383,E2 337.5752} C_DIS
LIN {X -40.0668,Y 100.0033,Z 112,A 106.6334,B 24.9293,C -1.9421,E1 24.9422,E2 339.068} C_DIS
LIN {X -36.339,Y 101.4175,Z 112,A 104.7401,B 24.9284,C -1.9536,E1 24.9471,E2 340.9379} C_DIS
LIN {X -33.9132,Y 102.2538,Z 112,A 102.561,B 24.9306,C -1.9242,E1 24.9531,E2 343.1911} C_DIS
LIN {X -29.544,Y 103.5994,Z 112,A 100.7998,B 24.9285,C -1.9525,E1 24.9576,E2 344.8879} C_DIS
LIN {X -25.6975,Y 104.6199,Z 112,A 98.7534,B 24.9282,C -1.9573,E1 24.9631,E2 346.9259} C_DIS
LIN {X -22.8451,Y 105.2795,Z 112,A 97.1716,B 24.9282,C -1.9577,E1 24.9674,E2 348.5087} C_DIS
LIN {X -16.8851,Y 106.399,Z 112,A 94.1297,B 24.9274,C -1.9673,E1 24.9758,E2 351.5309} C_DIS
LIN {X -14.1705,Y 106.794,Z 112,A 92.4582,B 24.928,C -1.9599,E1 24.9804,E2 353.2213} C_DIS
LIN {X -10.8889,Y 107.1784,Z 112,A 90.6218,B 24.9281,C -1.9578,E1 24.9855,E2 355.0638} C_DIS
LIN {X -7.184,Y 107.4898,Z 112,A 88.7551,B 24.9278,C -1.963,E1 24.9907,E2 356.919} C_DIS
LIN {X -4.2717,Y 107.6454,Z 112,A 87.0713,B 24.9281,C -1.9583,E1 24.9954,E2 358.6142} C_DIS
LIN {X -0.6047,Y 107.7279,Z 112,A 85.2218,B 24.9278,C -1.9628,E1 25.0006,E2 360.4532} C_DIS
LIN {X 3.3946,Y 107.6761,Z 112,A 83.0413,B 24.9279,C -1.961,E1 25.0067,E2 362.6377} C_DIS
LIN {X 6.7098,Y 107.5219,Z 112,A 81.2364,B 24.928,C -1.9594,E1 25.0117,E2 364.4457} C_DIS
LIN {X 10.1973,Y 107.2463,Z 112,A 79.3704,B 24.928,C -1.959,E1 25.0169,E2 366.3115} C_DIS
LIN {X 13.9181,Y 106.8267,Z 112,A 77.4071,B 24.928,C -1.9598,E1 25.0223,E2 368.2715} C_DIS
LIN {X 19.929,Y 105.8709,Z 112,A 74.453,B 24.9272,C -1.97,E1 25.0304,E2 371.1983} C_DIS
LIN {X 23.9897,Y 105.0249,Z 112,A 72.127,B 24.9277,C -1.9641,E1 25.0368,E2 373.5353} C_DIS
LIN {X 27.2334,Y 104.2314,Z 112,A 70.3102,B 24.9279,C -1.9614,E1 25.0417,E2 375.3559} C_DIS
LIN {X 29.6287,Y 103.5755,Z 112,A 68.998,B 24.9279,C -1.9608,E1 25.0452,E2 376.6672} C_DIS
LIN {X 32.6181,Y 102.6745,Z 112,A 67.4214,B 24.9278,C -1.9629,E1 25.0494,E2 378.236} C_DIS
LIN {X 35.1254,Y 101.844,Z 112,A 65.7406,B 24.9287,C -1.9505,E1 25.0539,E2 379.943} C_DIS
LIN {X 37.9993,Y 100.8055,Z 112,A 64.2437,B 24.9284,C -1.9542,E1 25.0578,E2 381.4278} C_DIS
LIN {X 41.1825,Y 99.5492,Z 112,A 62.5424,B 24.9282,C -1.9572,E1 25.0622,E2 383.1184} C_DIS
LIN {X 43.4507,Y 98.5794,Z 112,A 60.9106,B 24.9292,C -1.9426,E1 25.0665,E2 384.7806} C_DIS
LIN {X 47.6962,Y 96.5958,Z 112,A 58.6459,B 24.9288,C -1.9489,E1 25.0721,E2 387.0244} C_DIS
LIN {X 50.7995,Y 95.0026,Z 112,A 56.6465,B 24.9294,C -1.9405,E1 25.0771,E2 389.0382} C_DIS
LIN {X 53.7087,Y 93.3865,Z 112,A 55.0221,B 24.9291,C -1.944,E1 25.081,E2 390.6494} C_DIS
LIN {X 56.7033,Y 91.6002,Z 112,A 52.5415,B 24.9312,C -1.9154,E1 25.087,E2 393.1899} C_DIS
LIN {X 60.3399,Y 89.2455,Z 112,A 50.9431,B 24.9294,C -1.9408,E1 25.0906,E2 394.7229} C_DIS
LIN {X 62.8931,Y 87.4658,Z 112,A 49.1798,B 24.9299,C -1.9334,E1 25.0946,E2 396.4975} C_DIS
LIN {X 66.796,Y 84.5219,Z 112,A 46.7015,B 24.9299,C -1.9338,E1 25.1001,E2 398.9658} C_DIS
LIN {X 69.5275,Y 82.2909,Z 112,A 44.745,B 24.9304,C -1.9268,E1 25.1043,E2 400.9313} C_DIS
LIN {X 72.0562,Y 80.0852,Z 112,A 43.0371,B 24.9304,C -1.9265,E1 25.1079,E2 402.6333} C_DIS
LIN {X 74.8295,Y 77.4998,Z 112,A 41.0267,B 24.9307,C -1.9226,E1 25.112,E2 404.6447} C_DIS
LIN {X 77.2296,Y 75.1099,Z 112,A 39.1576,B 24.9312,C -1.9158,E1 25.1157,E2 406.5218} C_DIS
LIN {X 79.8572,Y 72.3108,Z 112,A 37.0729,B 24.9317,C -1.9094,E1 25.1196,E2 408.6124} C_DIS
LIN {X 82.1387,Y 69.7061,Z 112,A 34.788,B 24.9333,C -1.8865,E1 25.1238,E2 410.9411} C_DIS
LIN {X 84.6725,Y 66.6054,Z 112,A 33.3752,B 24.9315,C -1.9116,E1 25.1262,E2 412.2879} C_DIS
LIN {X 86.3753,Y 64.3827,Z 112,A 31.7982,B 24.932,C -1.9042,E1 25.1289,E2 413.8749} C_DIS
LIN {X 89.1175,Y 60.5289,Z 112,A 29.5301,B 24.9317,C -1.9084,E1 25.1325,E2 416.122} C_DIS
LIN {X 90.2524,Y 58.8259,Z 112,A 28.2645,B 24.9325,C -1.898,E1 25.1344,E2 417.4059} C_DIS
LIN {X 92.3649,Y 55.4502,Z 112,A 25.8915,B 24.9336,C -1.8815,E1 25.138,E2 419.8058} C_DIS
LIN {X 94.2915,Y 52.1057,Z 112,A 23.9768,B 24.9336,C -1.8818,E1 25.1406,E2 421.7098} C_DIS
LIN {X 95.9569,Y 48.9688,Z 112,A 22.1593,B 24.9338,C -1.8796,E1 25.1429,E2 423.5228} C_DIS
LIN {X 97.6956,Y 45.4009,Z 112,A 20.0734,B 24.9341,C -1.8747,E1 25.1454,E2 425.6091} C_DIS
LIN {X 98.8431,Y 42.8457,Z 112,A 18.6695,B 24.9341,C -1.8741,E1 25.147,E2 427.0067} C_DIS
LIN {X 99.8245,Y 40.5062,Z 112,A 17.2306,B 24.9347,C -1.8663,E1 25.1485,E2 428.4562} C_DIS
LIN {X 101.2213,Y 36.877,Z 112,A 15.1198,B 24.9353,C -1.8583,E1 25.1506,E2 430.574} C_DIS
LIN {X 102.2476,Y 33.9316,Z 112,A 13.4202,B 24.9357,C -1.8516,E1 25.1521,E2 432.2799} C_DIS
LIN {X 103.442,Y 30.0953,Z 112,A 11.4827,B 24.9356,C -1.8537,E1 25.1537,E2 434.2014} C_DIS
LIN {X 104.1429,Y 27.5717,Z 112,A 10.0987,B 24.9359,C -1.8498,E1 25.1547,E2 435.5866} C_DIS
LIN {X 105.0371,Y 23.9368,Z 112,A 8.0958,B 24.9363,C -1.8431,E1 25.156,E2 437.5938} C_DIS
LIN {X 105.7801,Y 20.4016,Z 112,A 6.1007,B 24.937,C -1.8339,E1 25.1571,E2 439.5989} C_DIS
LIN {X 106.3636,Y 17.114,Z 112,A 4.2366,B 24.9376,C -1.8244,E1 25.158,E2 441.4745} C_DIS
LIN {X 106.8562,Y 13.691,Z 112,A 2.505,B 24.9376,C -1.8232,E1 25.1587,E2 443.1985} C_DIS
LIN {X 107.2716,Y 9.9231,Z 112,A 0.5163,B 24.9381,C -1.818,E1 25.1592,E2 445.1879} C_DIS
LIN {X 107.5158,Y 6.7997,Z 112,A -1.2147,B 24.9386,C -1.8098,E1 25.1596,E2 446.9279} C_DIS
LIN {X 107.6916,Y 2.8914,Z 112,A -3.1315,B 24.9386,C -1.8102,E1 25.1598,E2 448.8324} C_DIS
LIN {X 107.7287,Y -0.5801,Z 112,A -5.0638,B 24.9392,C -1.8005,E1 25.1598,E2 450.7761} C_DIS
LIN {X 107.6604,Y -3.9061,Z 112,A -6.8942,B 24.9398,C -1.792,E1 25.1596,E2 452.6155} C_DIS
LIN {X 107.4321,Y -8.02,Z 112,A -9.0379,B 24.9401,C -1.787,E1 25.1592,E2 454.7584} C_DIS
LIN {X 107.1125,Y -11.5177,Z 112,A -10.9151,B 24.9406,C -1.7805,E1 25.1587,E2 456.6397} C_DIS
LIN {X 106.312,Y -17.4224,Z 112,A -14.6567,B 24.9429,C -1.7455,E1 25.1571,E2 460.4419} C_DIS
LIN {X 105.4788,Y -21.9074,Z 112,A -16.1992,B 24.9409,C -1.776,E1 25.1563,E2 461.9035} C_DIS
LIN {X 104.5833,Y -25.8476,Z 112,A -18.4528,B 24.9416,C -1.7645,E1 25.1549,E2 464.1711} C_DIS
LIN {X 103.6244,Y -29.456,Z 112,A -20.5519,B 24.9424,C -1.7532,E1 25.1533,E2 466.2847} C_DIS
LIN {X 102.6988,Y -32.5428,Z 112,A -22.0867,B 24.9422,C -1.7556,E1 25.1521,E2 467.8053} C_DIS
LIN {X 101.7012,Y -35.5324,Z 112,A -23.8958,B 24.943,C -1.7446,E1 25.1504,E2 469.6301} C_DIS
LIN {X 100.1972,Y -39.5754,Z 112,A -26.1407,B 24.9433,C -1.7396,E1 25.1482,E2 471.8743} C_DIS
LIN {X 99.0778,Y -42.3026,Z 112,A -27.993,B 24.9444,C -1.7224,E1 25.1462,E2 473.7569} C_DIS
LIN {X 96.9898,Y -46.8904,Z 112,A -30.3873,B 24.9441,C -1.7267,E1 25.1433,E2 476.1282} C_DIS
LIN {X 95.2308,Y -50.3665,Z 112,A -32.4761,B 24.9446,C -1.7198,E1 25.1407,E2 478.2222} C_DIS
LIN {X 93.6797,Y -53.1985,Z 112,A -34.2171,B 24.945,C -1.7137,E1 25.1383,E2 479.9686} C_DIS
LIN {X 91.6569,Y -56.612,Z 112,A -36.0967,B 24.9447,C -1.7176,E1 25.1356,E2 481.8293} C_DIS
LIN {X 89.2147,Y -60.3855,Z 112,A -38.1864,B 24.9443,C -1.7239,E1 25.1325,E2 483.8938} C_DIS
LIN {X 87.8165,Y -62.4016,Z 112,A -39.919,B 24.9457,C -1.7017,E1 25.1296,E2 485.6703} C_DIS
LIN {X 84.1519,Y -67.2642,Z 112,A -42.974,B 24.9457,C -1.7007,E1 25.1245,E2 488.7129} C_DIS
LIN {X 80.4766,Y -71.619,Z 112,A -45.8588,B 24.9459,C -1.6991,E1 25.1193,E2 491.5885} C_DIS
LIN {X 76.0709,Y -76.2833,Z 112,A -49.6959,B 24.9476,C -1.6722,E1 25.1118,E2 495.4724} C_DIS
LIN {X 72.2811,Y -79.8838,Z 112,A -52.1419,B 24.9471,C -1.6799,E1 25.1068,E2 497.8903} C_DIS
LIN {X 67.3765,Y -84.0619,Z 112,A -55.8365,B 24.9483,C -1.6607,E1 25.0989,E2 501.616} C_DIS
LIN {X 64.7194,Y -86.1224,Z 112,A -57.4465,B 24.9481,C -1.6645,E1 25.0953,E2 503.2113} C_DIS
LIN {X 62.0362,Y -88.0773,Z 112,A -59.6606,B 24.9495,C -1.6418,E1 25.0902,E2 505.4713} C_DIS
LIN {X 59.2432,Y -89.9773,Z 112,A -60.8849,B 24.9482,C -1.6625,E1 25.0874,E2 506.6426} C_DIS
LIN {X 56.6244,Y -91.6494,Z 112,A -62.7772,B 24.949,C -1.6491,E1 25.0829,E2 508.5604} C_DIS
LIN {X 53.1899,Y -93.6846,Z 112,A -64.6671,B 24.9487,C -1.6551,E1 25.0784,E2 510.4305} C_DIS
LIN {X 49.3985,Y -95.7373,Z 112,A -66.8501,B 24.9487,C -1.6557,E1 25.073,E2 512.6057} C_DIS
LIN {X 45.7949,Y -97.5122,Z 112,A -69.6054,B 24.9504,C -1.6263,E1 25.0659,E2 515.4233} C_DIS
LIN {X 42.6578,Y -98.925,Z 112,A -70.9303,B 24.9493,C -1.6447,E1 25.0627,E2 516.7016} C_DIS
LIN {X 39.0669,Y -100.397,Z 112,A -72.893,B 24.9493,C -1.646,E1 25.0576,E2 518.6567} C_DIS
LIN {X 36.3498,Y -101.4136,Z 112,A -74.7243,B 24.9501,C -1.6318,E1 25.0527,E2 520.5177} C_DIS
LIN {X 32.4645,Y -102.7232,Z 112,A -76.6553,B 24.9496,C -1.6395,E1 25.0477,E2 522.4268} C_DIS
LIN {X 29.6494,Y -103.5696,Z 112,A -78.6739,B 24.9509,C -1.6189,E1 25.0421,E2 524.4907} C_DIS
LIN {X 23.6684,Y -105.0991,Z 112,A -81.5271,B 24.95,C -1.6334,E1 25.0345,E2 527.3055} C_DIS
LIN {X 21.1388,Y -105.6366,Z 112,A -83.2262,B 24.9509,C -1.6189,E1 25.0298,E2 529.0369} C_DIS
LIN {X 16.421,Y -106.4707,Z 112,A -85.552,B 24.9505,C -1.6261,E1 25.0234,E2 531.3433} C_DIS
LIN {X 13.4652,Y -106.8854,Z 112,A -87.1868,B 24.9506,C -1.6231,E1 25.0189,E2 532.9838} C_DIS
LIN {X 9.8008,Y -107.2829,Z 112,A -89.0597,B 24.9505,C -1.6256,E1 25.0137,E2 534.8496} C_DIS
LIN {X 5.9961,Y -107.5626,Z 112,A -91.1128,B 24.9505,C -1.6237,E1 25.0079,E2 536.9063} C_DIS
LIN {X 2.8488,Y -107.6929,Z 112,A -92.6676,B 24.9503,C -1.628,E1 25.0036,E2 538.4505} C_DIS
LIN {X 0.7561,Y -107.7252,Z 112,A -93.3382,B 24.9492,C -1.6458,E1 25.0019,E2 539.0788} C_DIS
Enddeposition()
LIN {X 0.7561,Y -107.7252,Z 112,A -93.3382,B 24.9492,C -1.6458,E1 25.0019,E2 539.0788} C_DIS
Startdeposition()
$VEL.CP = VEL_PRINT
LIN {X 1.3128,Y -106.7926,Z 112,A -92.8945,B 24.9479,C -1.6679,E1 25.0033,E2 538.5827} C_DIS
LIN {X 3.8389,Y -106.7312,Z 112,A -91.536,B 24.9479,C -1.6685,E1 25.0071,E2 537.2232} C_DIS
LIN {X 6.4508,Y -106.6052,Z 112,A -90.1341,B 24.9478,C -1.6691,E1 25.011,E2 535.8205} C_DIS
LIN {X 9.852,Y -106.3433,Z 112,A -88.27,B 24.9477,C -1.6714,E1 25.0162,E2 533.9519} C_DIS
LIN {X 13.0717,Y -105.9977,Z 112,A -86.5739,B 24.9477,C -1.6707,E1 25.0209,E2 532.2586} C_DIS
LIN {X 15.5775,Y -105.658,Z 112,A -85.2166,B 24.9477,C -1.6717,E1 25.0246,E2 530.9002} C_DIS
LIN {X 18.1613,Y -105.2447,Z 112,A -83.8149,B 24.9476,C -1.6727,E1 25.0285,E2 529.4976} C_DIS
LIN {X 20.3762,Y -104.837,Z 112,A -82.5515,B 24.9474,C -1.676,E1 25.032,E2 528.2278} C_DIS
LIN {X 24.5467,Y -103.9408,Z 112,A -80.3292,B 24.9474,C -1.6753,E1 25.038,E2 526.01} C_DIS
LIN {X 27.1149,Y -103.3007,Z 112,A -78.9172,B 24.9474,C -1.6765,E1 25.0418,E2 524.5975} C_DIS
LIN {X 29.4253,Y -102.6656,Z 112,A -77.6562,B 24.9474,C -1.6769,E1 25.0452,E2 523.3375} C_DIS
LIN {X 32.0439,Y -101.879,Z 112,A -76.1559,B 24.9471,C -1.68,E1 25.0492,E2 521.8326} C_DIS
LIN {X 34.652,Y -101.0223,Z 112,A -74.6938,B 24.9471,C -1.6814,E1 25.0531,E2 520.37} C_DIS
LIN {X 37.1996,Y -100.1128,Z 112,A -73.2495,B 24.9469,C -1.683,E1 25.0569,E2 518.9248} C_DIS
LIN {X 39.5554,Y -99.205,Z 112,A -71.9329,B 24.9469,C -1.6833,E1 25.0603,E2 517.6104} C_DIS
LIN {X 43.1971,Y -97.6744,Z 112,A -69.7749,B 24.9466,C -1.6881,E1 25.0659,E2 515.4462} C_DIS
LIN {X 45.5919,Y -96.5799,Z 112,A -68.3791,B 24.9466,C -1.6896,E1 25.0694,E2 514.0504} C_DIS
LIN {X 48.015,Y -95.3989,Z 112,A -66.9381,B 24.9464,C -1.6918,E1 25.073,E2 512.6082} C_DIS
LIN {X 50.2488,Y -94.2408,Z 112,A -65.5932,B 24.9462,C -1.6939,E1 25.0763,E2 511.2621} C_DIS
LIN {X 52.1686,Y -93.1902,Z 112,A -64.3464,B 24.9459,C -1.6991,E1 25.0794,E2 510.0066} C_DIS
LIN {X 54.9017,Y -91.6089,Z 112,A -62.7365,B 24.9459,C -1.6986,E1 25.0833,E2 508.4028} C_DIS
LIN {X 57.0518,Y -90.2849,Z 112,A -61.3838,B 24.9458,C -1.7011,E1 25.0865,E2 507.0485} C_DIS
LIN {X 59.2447,Y -88.8613,Z 112,A -59.9803,B 24.9456,C -1.704,E1 25.0898,E2 505.6429} C_DIS
LIN {X 61.5008,Y -87.3157,Z 112,A -58.5319,B 24.9454,C -1.7061,E1 25.0931,E2 504.1944} C_DIS
LIN {X 64.6551,Y -85.0064,Z 112,A -56.4421,B 24.9452,C -1.7103,E1 25.0978,E2 502.1023} C_DIS
LIN {X 66.6736,Y -83.4321,Z 112,A -55.0739,B 24.945,C -1.7131,E1 25.1008,E2 500.7326} C_DIS
LIN {X 68.6845,Y -81.7846,Z 112,A -53.4932,B 24.9443,C -1.7242,E1 25.1042,E2 499.1317} C_DIS
LIN {X 71.2638,Y -79.5452,Z 112,A -51.7725,B 24.9443,C -1.7237,E1 25.1078,E2 497.419} C_DIS
LIN {X 73.5537,Y -77.4345,Z 112,A -50.0249,B 24.9438,C -1.7309,E1 25.1114,E2 495.6614} C_DIS
LIN {X 76.2998,Y -74.7296,Z 112,A -47.9381,B 24.9435,C -1.7368,E1 25.1155,E2 493.5695} C_DIS
LIN {X 78.6745,Y -72.2239,Z 112,A -46.296,B 24.9437,C -1.7325,E1 25.1186,E2 491.945} C_DIS
LIN {X 80.4265,Y -70.2677,Z 112,A -44.8959,B 24.9435,C -1.7357,E1 25.1212,E2 490.5435} C_DIS
LIN {X 82.4653,Y -67.8653,Z 112,A -43.0377,B 24.9428,C -1.7474,E1 25.1245,E2 488.6662} C_DIS
LIN {X 84.7378,Y -65.004,Z 112,A -41.2398,B 24.9428,C -1.7457,E1 25.1276,E2 486.8809} C_DIS
LIN {X 86.5057,Y -62.6343,Z 112,A -39.6947,B 24.9428,C -1.7482,E1 25.1301,E2 485.3371} C_DIS
LIN {X 88.0094,Y -60.503,Z 112,A -38.3038,B 24.9425,C -1.7518,E1 25.1324,E2 483.9447} C_DIS
LIN {X 89.5095,Y -58.2616,Z 112,A -36.8664,B 24.9422,C -1.7555,E1 25.1346,E2 482.5058} C_DIS
LIN {X 90.8225,Y -56.1913,Z 112,A -35.5437,B 24.942,C -1.7596,E1 25.1365,E2 481.18} C_DIS
LIN {X 92.2283,Y -53.8537,Z 112,A -34.104,B 24.9418,C -1.7628,E1 25.1386,E2 479.7402} C_DIS
LIN {X 93.5195,Y -51.5788,Z 112,A -32.7068,B 24.9415,C -1.7667,E1 25.1405,E2 478.3411} C_DIS
LIN {X 94.7965,Y -49.1935,Z 112,A -31.2658,B 24.9412,C -1.7705,E1 25.1424,E2 476.8987} C_DIS
LIN {X 95.9378,Y -46.9278,Z 112,A -29.9123,B 24.941,C -1.7743,E1 25.1441,E2 475.5435} C_DIS
LIN {X 97.0934,Y -44.4887,Z 112,A -28.4771,B 24.9407,C -1.7781,E1 25.1457,E2 474.107} C_DIS
LIN {X 98.1506,Y -42.1048,Z 112,A -27.0871,B 24.9405,C -1.782,E1 25.1473,E2 472.7154} C_DIS
LIN {X 99.1709,Y -39.6421,Z 112,A -25.6675,B 24.9402,C -1.786,E1 25.1488,E2 471.2943} C_DIS
LIN {X 100.0803,Y -37.2858,Z 112,A -24.3202,B 24.94,C -1.7899,E1 25.1501,E2 469.9454} C_DIS
LIN {X 100.9634,Y -34.8235,Z 112,A -22.9225,B 24.9397,C -1.794,E1 25.1514,E2 468.5457} C_DIS
LIN {X 101.752,Y -32.4453,Z 112,A -21.5837,B 24.9394,C -1.798,E1 25.1526,E2 467.205} C_DIS
LIN {X 102.5732,Y -29.751,Z 112,A -20.0902,B 24.9391,C -1.802,E1 25.1538,E2 465.7106} C_DIS
LIN {X 103.2711,Y -27.2299,Z 112,A -18.6969,B 24.9389,C -1.8061,E1 25.1548,E2 464.3158} C_DIS
LIN {X 103.9069,Y -24.6928,Z 112,A -17.3001,B 24.9386,C -1.8103,E1 25.1557,E2 462.9171} C_DIS
LIN {X 104.7274,Y -20.9387,Z 112,A -15.2527,B 24.9382,C -1.8163,E1 25.1569,E2 460.8674} C_DIS
LIN {X 105.2055,Y -18.3856,Z 112,A -13.8685,B 24.9379,C -1.8204,E1 25.1576,E2 459.4817} C_DIS
LIN {X 105.6202,Y -15.8294,Z 112,A -12.4879,B 24.9376,C -1.8245,E1 25.1582,E2 458.0995} C_DIS
LIN {X 106.0653,Y -12.4946,Z 112,A -10.6397,B 24.9371,C -1.8323,E1 25.1588,E2 456.2438} C_DIS
LIN {X 106.4075,Y -9.1562,Z 112,A -8.912,B 24.9369,C -1.8349,E1 25.1593,E2 454.5201} C_DIS
LIN {X 106.594,Y -6.6345,Z 112,A -7.5648,B 24.9366,C -1.839,E1 25.1595,E2 453.1715} C_DIS
LIN {X 106.7244,Y -4.0217,Z 112,A -6.1682,B 24.9363,C -1.8432,E1 25.1597,E2 451.7731} C_DIS
LIN {X 106.7926,Y -1.3139,Z 112,A -4.7532,B 24.9361,C -1.8463,E1 25.1597,E2 450.3594} C_DIS
LIN {X 106.7701,Y 2.5379,Z 112,A -2.676,B 24.9356,C -1.8534,E1 25.1597,E2 448.2777} C_DIS
LIN {X 106.6719,Y 5.2438,Z 112,A -1.235,B 24.9353,C -1.8576,E1 25.1595,E2 446.8353} C_DIS
LIN {X 106.5114,Y 7.8557,Z 112,A 0.1607,B 24.935,C -1.8618,E1 25.1593,E2 445.4381} C_DIS
LIN {X 106.2328,Y 10.9811,Z 112,A 1.9062,B 24.9345,C -1.8699,E1 25.1588,E2 443.6838} C_DIS
LIN {X 105.8285,Y 14.3776,Z 112,A 3.6531,B 24.9343,C -1.8719,E1 25.1582,E2 441.9425} C_DIS
LIN {X 105.4445,Y 16.9662,Z 112,A 5.0495,B 24.934,C -1.876,E1 25.1576,E2 440.5446} C_DIS
LIN {X 104.9971,Y 19.5445,Z 112,A 6.4437,B 24.9337,C -1.88,E1 25.1569,E2 439.1491} C_DIS
LIN {X 104.4868,Y 22.111,Z 112,A 7.8345,B 24.9335,C -1.8839,E1 25.1561,E2 437.7574} C_DIS
LIN {X 103.6181,Y 25.8763,Z 112,A 9.9029,B 24.933,C -1.8901,E1 25.1548,E2 435.6862} C_DIS
LIN {X 102.9552,Y 28.399,Z 112,A 11.2874,B 24.9328,C -1.8938,E1 25.1538,E2 434.3011} C_DIS
LIN {X 102.2308,Y 30.9051,Z 112,A 12.6772,B 24.9325,C -1.8976,E1 25.1527,E2 432.9101} C_DIS
LIN {X 101.4376,Y 33.4172,Z 112,A 14.082,B 24.9322,C -1.9015,E1 25.1515,E2 431.504} C_DIS
LIN {X 100.559,Y 35.976,Z 112,A 15.5236,B 24.9319,C -1.9054,E1 25.1501,E2 430.0613} C_DIS
LIN {X 99.6479,Y 38.4275,Z 112,A 16.9133,B 24.9317,C -1.909,E1 25.1488,E2 428.6709} C_DIS
LIN {X 98.1619,Y 42.0789,Z 112,A 19.02,B 24.9313,C -1.9148,E1 25.1465,E2 426.5622} C_DIS
LIN {X 97.1007,Y 44.473,Z 112,A 20.416,B 24.931,C -1.9185,E1 25.1449,E2 425.1651} C_DIS
LIN {X 96.0136,Y 46.7726,Z 112,A 21.7777,B 24.9307,C -1.9222,E1 25.1433,E2 423.8019} C_DIS
LIN {X 94.9916,Y 48.812,Z 112,A 23.0299,B 24.9304,C -1.9269,E1 25.1417,E2 422.5454} C_DIS
LIN {X 93.6111,Y 51.4125,Z 112,A 24.5621,B 24.9302,C -1.9292,E1 25.1396,E2 421.0158} C_DIS
LIN {X 92.2808,Y 53.7646,Z 112,A 26.0005,B 24.93,C -1.9326,E1 25.1376,E2 419.5767} C_DIS
LIN {X 90.2786,Y 57.0618,Z 112,A 28.0611,B 24.9296,C -1.9377,E1 25.1346,E2 417.5145} C_DIS
LIN {X 88.8529,Y 59.2574,Z 112,A 29.4578,B 24.9294,C -1.941,E1 25.1325,E2 416.117} C_DIS
LIN {X 87.4551,Y 61.3004,Z 112,A 30.7966,B 24.9291,C -1.9449,E1 25.1303,E2 414.7756} C_DIS
LIN {X 85.9759,Y 63.3578,Z 112,A 32.1588,B 24.9288,C -1.9484,E1 25.1281,E2 413.4117} C_DIS
LIN {X 84.2045,Y 65.6961,Z 112,A 33.8895,B 24.9281,C -1.9589,E1 25.1251,E2 411.6643} C_DIS
LIN {X 82.156,Y 68.2375,Z 112,A 35.4987,B 24.9281,C -1.9571,E1 25.1223,E2 410.067} C_DIS
LIN {X 79.8348,Y 70.9402,Z 112,A 37.4564,B 24.9277,C -1.9634,E1 25.1187,E2 408.1031} C_DIS
LIN {X 77.7962,Y 73.1691,Z 112,A 38.9383,B 24.9279,C -1.9612,E1 25.1159,E2 406.633} C_DIS
LIN {X 76.0111,Y 75.0219,Z 112,A 40.3349,B 24.9276,C -1.9649,E1 25.1131,E2 405.2336} C_DIS
LIN {X 74.1489,Y 76.8629,Z 112,A 41.7333,B 24.9274,C -1.9676,E1 25.1103,E2 403.8347} C_DIS
LIN {X 72.2429,Y 78.6571,Z 112,A 43.1314,B 24.9272,C -1.9702,E1 25.1075,E2 402.436} C_DIS
LIN {X 70.0013,Y 80.6591,Z 112,A 44.7991,B 24.9268,C -1.9757,E1 25.104,E2 400.7619} C_DIS
LIN {X 67.2782,Y 82.9434,Z 112,A 46.636,B 24.9268,C -1.9764,E1 25.1,E2 398.9303} C_DIS
LIN {X 65.1412,Y 84.6321,Z 112,A 48.1624,B 24.9264,C -1.9819,E1 25.0967,E2 397.3968} C_DIS
LIN {X 63.0105,Y 86.2302,Z 112,A 49.574,B 24.9262,C -1.9836,E1 25.0935,E2 395.986} C_DIS
LIN {X 60.5049,Y 88.0081,Z 112,A 51.146,B 24.9262,C -1.9832,E1 25.0899,E2 394.4204} C_DIS
LIN {X 58.2644,Y 89.5076,Z 112,A 52.5866,B 24.9261,C -1.9853,E1 25.0865,E2 392.9796} C_DIS
LIN {X 56.0658,Y 90.9008,Z 112,A 53.9716,B 24.926,C -1.987,E1 25.0833,E2 391.595} C_DIS
LIN {X 53.8595,Y 92.2249,Z 112,A 55.3553,B 24.9258,C -1.9892,E1 25.0799,E2 390.2104} C_DIS
LIN {X 51.5839,Y 93.5167,Z 112,A 56.7364,B 24.9258,C -1.9902,E1 25.0766,E2 388.8309} C_DIS
LIN {X 49.183,Y 94.802,Z 112,A 58.2102,B 24.9255,C -1.9927,E1 25.0729,E2 387.3555} C_DIS
LIN {X 46.9297,Y 95.9368,Z 112,A 59.5644,B 24.9255,C -1.9944,E1 25.0695,E2 386.0007} C_DIS
LIN {X 44.4876,Y 97.0939,Z 112,A 61.0069,B 24.9253,C -1.9959,E1 25.0659,E2 384.5585} C_DIS
LIN {X 42.0786,Y 98.162,Z 112,A 62.418,B 24.9252,C -1.9973,E1 25.0623,E2 383.1474} C_DIS
LIN {X 39.661,Y 99.1635,Z 112,A 63.8186,B 24.9252,C -1.9987,E1 25.0587,E2 381.7468} C_DIS
LIN {X 37.3017,Y 100.0743,Z 112,A 65.1724,B 24.925,C -1.9998,E1 25.0551,E2 380.3931} C_DIS
LIN {X 34.8237,Y 100.9634,Z 112,A 66.5858,B 24.925,C -2.0011,E1 25.0514,E2 378.9795} C_DIS
LIN {X 32.2552,Y 101.8135,Z 112,A 68.0312,B 24.9248,C -2.0021,E1 25.0476,E2 377.5347} C_DIS
LIN {X 29.7523,Y 102.5728,Z 112,A 69.4323,B 24.9248,C -2.003,E1 25.0438,E2 376.1337} C_DIS
LIN {X 27.2318,Y 103.2705,Z 112,A 70.8329,B 24.9248,C -2.0038,E1 25.04,E2 374.7335} C_DIS
LIN {X 24.6875,Y 103.9082,Z 112,A 72.2387,B 24.9247,C -2.0046,E1 25.0362,E2 373.3279} C_DIS
LIN {X 22.1424,Y 104.48,Z 112,A 73.6335,B 24.9247,C -2.0051,E1 25.0324,E2 371.9337} C_DIS
LIN {X 19.6676,Y 104.9735,Z 112,A 75.1138,B 24.9242,C -2.0108,E1 25.0283,E2 370.4417} C_DIS
LIN {X 15.6752,Y 105.6441,Z 112,A 77.1597,B 24.9245,C -2.0064,E1 25.0227,E2 368.4082} C_DIS
LIN {X 13.1716,Y 105.9848,Z 112,A 78.5147,B 24.9245,C -2.0067,E1 25.019,E2 367.0536} C_DIS
LIN {X 9.6731,Y 106.3598,Z 112,A 80.4728,B 24.9243,C -2.0098,E1 25.0135,E2 365.0895} C_DIS
LIN {X 6.64,Y 106.5936,Z 112,A 82.0366,B 24.9245,C -2.0071,E1 25.0092,E2 363.5328} C_DIS
LIN {X 4.0265,Y 106.7242,Z 112,A 83.4408,B 24.9245,C -2.007,E1 25.0052,E2 362.1291} C_DIS
LIN {X 1.3207,Y 106.7925,Z 112,A 84.89,B 24.9245,C -2.0067,E1 25.0012,E2 360.6809} C_DIS
LIN {X -0.7435,Y 106.7962,Z 112,A 86.0727,B 24.9243,C -2.0095,E1 24.9979,E2 359.4915} C_DIS
LIN {X -3.8433,Y 106.731,Z 112,A 87.6653,B 24.9245,C -2.0062,E1 24.9935,E2 357.9066} C_DIS
LIN {X -6.4571,Y 106.6048,Z 112,A 89.0533,B 24.9246,C -2.005,E1 24.9896,E2 356.521} C_DIS
LIN {X -9.0681,Y 106.4145,Z 112,A 90.4735,B 24.9246,C -2.005,E1 24.9856,E2 355.1002} C_DIS
LIN {X -11.6723,Y 106.1604,Z 112,A 91.8818,B 24.9246,C -2.0044,E1 24.9817,E2 353.6923} C_DIS
LIN {X -15.5801,Y 105.6577,Z 112,A 93.9984,B 24.9248,C -2.0032,E1 24.9759,E2 351.5771} C_DIS
LIN {X -18.2013,Y 105.238,Z 112,A 95.4345,B 24.9248,C -2.0027,E1 24.9719,E2 350.1409} C_DIS
LIN {X -20.765,Y 104.7622,Z 112,A 96.8307,B 24.9248,C -2.0014,E1 24.9681,E2 348.7461} C_DIS
LIN {X -23.3182,Y 104.2236,Z 112,A 98.2258,B 24.925,C -2,E1 24.9643,E2 347.3527} C_DIS
LIN {X -25.8583,Y 103.6225,Z 112,A 99.632,B 24.925,C -1.9989,E1 24.9605,E2 345.9471} C_DIS
LIN {X -28.2986,Y 102.9824,Z 112,A 100.9911,B 24.9252,C -1.9977,E1 24.9568,E2 344.5887} C_DIS
LIN {X -30.8886,Y 102.2357,Z 112,A 102.4387,B 24.9252,C -1.9962,E1 24.9529,E2 343.1423} C_DIS
LIN {X -33.3733,Y 101.4518,Z 112,A 103.8049,B 24.9255,C -1.9933,E1 24.9493,E2 341.7805} C_DIS
LIN {X -35.978,Y 100.5583,Z 112,A 105.318,B 24.9255,C -1.9928,E1 24.9453,E2 340.2656} C_DIS
LIN {X -38.4309,Y 99.6466,Z 112,A 106.7258,B 24.9257,C -1.9911,E1 24.9417,E2 338.859} C_DIS
LIN {X -40.7771,Y 98.7092,Z 112,A 108.0939,B 24.9257,C -1.9897,E1 24.9381,E2 337.4912} C_DIS
LIN {X -43.2002,Y 97.6731,Z 112,A 109.4762,B 24.926,C -1.9864,E1 24.9346,E2 336.1134} C_DIS
LIN {X -45.5706,Y 96.5898,Z 112,A 110.9065,B 24.926,C -1.9855,E1 24.931,E2 334.6817} C_DIS
LIN {X -47.7147,Y 95.5477,Z 112,A 112.2133,B 24.9262,C -1.9845,E1 24.9277,E2 333.3738} C_DIS
LIN {X -50.3023,Y 94.2126,Z 112,A 113.9537,B 24.9258,C -1.9887,E1 24.9234,E2 331.6188} C_DIS
LIN {X -53.3434,Y 92.5228,Z 112,A 115.6999,B 24.9264,C -1.9808,E1 24.9191,E2 329.8861} C_DIS
LIN {X -55.9478,Y 90.9732,Z 112,A 117.2639,B 24.9268,C -1.9755,E1 24.9154,E2 328.33} C_DIS
LIN {X -58.246,Y 89.5198,Z 112,A 118.726,B 24.927,C -1.9728,E1 24.912,E2 326.8695} C_DIS
LIN {X -60.4053,Y 88.077,Z 112,A 120.1283,B 24.9272,C -1.9704,E1 24.9088,E2 325.4684} C_DIS
LIN {X -62.5264,Y 86.584,Z 112,A 121.5682,B 24.9272,C -1.9694,E1 24.9055,E2 324.0258} C_DIS
LIN {X -65.1498,Y 84.6255,Z 112,A 123.3013,B 24.9276,C -1.9648,E1 24.9016,E2 322.2974} C_DIS
LIN {X -67.3521,Y 82.8835,Z 112,A 124.9264,B 24.9276,C -1.966,E1 24.8981,E2 320.6634} C_DIS
LIN {X -70.224,Y 80.4646,Z 112,A 126.8388,B 24.9281,C -1.9576,E1 24.894,E2 318.7635} C_DIS
LIN {X -72.2063,Y 78.6906,Z 112,A 128.2621,B 24.9284,C -1.9542,E1 24.8911,E2 317.3427} C_DIS
LIN {X -74.1437,Y 76.8679,Z 112,A 129.7711,B 24.9284,C -1.9539,E1 24.888,E2 315.8283} C_DIS
LIN {X -76.4287,Y 74.5991,Z 112,A 131.434,B 24.9289,C -1.9472,E1 24.8848,E2 314.1741} C_DIS
LIN {X -78.2231,Y 72.7151,Z 112,A 132.8373,B 24.9291,C -1.944,E1 24.8821,E2 312.7723} C_DIS
LIN {X -79.9793,Y 70.7789,Z 112,A 134.2482,B 24.9294,C -1.9408,E1 24.8795,E2 311.3628} C_DIS
LIN {X -81.7456,Y 68.7313,Z 112,A 135.8947,B 24.9291,C -1.9443,E1 24.8765,E2 309.7004} C_DIS
LIN {X -83.7824,Y 66.2304,Z 112,A 137.4621,B 24.9299,C -1.9337,E1 24.8738,E2 308.1509} C_DIS
LIN {X -85.7321,Y 63.689,Z 112,A 139.1755,B 24.9303,C -1.9288,E1 24.8709,E2 306.4409} C_DIS
LIN {X -87.2664,Y 61.5699,Z 112,A 140.5875,B 24.9305,C -1.9253,E1 24.8686,E2 305.0305} C_DIS
LIN {X -88.7483,Y 59.4139,Z 112,A 142.0026,B 24.9308,C -1.9218,E1 24.8664,E2 303.6167} C_DIS
LIN {X -90.1844,Y 57.2107,Z 112,A 143.4218,B 24.931,C -1.9181,E1 24.8643,E2 302.1991} C_DIS
LIN {X -91.6013,Y 54.9143,Z 112,A 144.8756,B 24.9313,C -1.9142,E1 24.8621,E2 300.7472} C_DIS
LIN {X -92.8289,Y 52.8106,Z 112,A 146.1962,B 24.9315,C -1.9109,E1 24.8603,E2 299.4275} C_DIS
LIN {X -94.0518,Y 50.5999,Z 112,A 147.5828,B 24.9317,C -1.9081,E1 24.8585,E2 298.0404} C_DIS
LIN {X -95.4069,Y 47.9988,Z 112,A 149.1277,B 24.9322,C -1.9023,E1 24.8565,E2 296.5008} C_DIS
LIN {X -96.5524,Y 45.6509,Z 112,A 150.5475,B 24.9324,C -1.8988,E1 24.8548,E2 295.0818} C_DIS
LIN {X -97.6036,Y 43.3569,Z 112,A 151.9155,B 24.9327,C -1.8952,E1 24.8532,E2 293.7148} C_DIS
LIN {X -98.6352,Y 40.9557,Z 112,A 153.3264,B 24.9329,C -1.8913,E1 24.8517,E2 292.3056} C_DIS
LIN {X -99.6406,Y 38.4463,Z 112,A 154.7832,B 24.9332,C -1.887,E1 24.8502,E2 290.8507} C_DIS
LIN {X -100.5205,Y 36.0818,Z 112,A 156.1462,B 24.9335,C -1.8832,E1 24.8489,E2 289.4891} C_DIS
LIN {X -101.4013,Y 33.528,Z 112,A 157.5985,B 24.9338,C -1.8787,E1 24.8476,E2 288.0391} C_DIS
LIN {X -102.1746,Y 31.0907,Z 112,A 158.9897,B 24.9341,C -1.8751,E1 24.8465,E2 286.6486} C_DIS
LIN {X -102.9352,Y 28.473,Z 112,A 160.4578,B 24.9344,C -1.8707,E1 24.8453,E2 285.1825} C_DIS
LIN {X -103.5793,Y 26.0312,Z 112,A 161.8278,B 24.9347,C -1.8669,E1 24.8444,E2 283.8134} C_DIS
LIN {X -104.2059,Y 23.3994,Z 112,A 163.2847,B 24.935,C -1.8625,E1 24.8435,E2 282.3586} C_DIS
LIN {X -104.7295,Y 20.9287,Z 112,A 164.6524,B 24.9352,C -1.8586,E1 24.8427,E2 280.9921} C_DIS
LIN {X -105.2105,Y 18.358,Z 112,A 166.0656,B 24.9355,C -1.8545,E1 24.842,E2 279.5805} C_DIS
LIN {X -105.6284,Y 15.7767,Z 112,A 167.4547,B 24.9359,C -1.8494,E1 24.8414,E2 278.1951} C_DIS
LIN {X -105.9498,Y 13.442,Z 112,A 168.7533,B 24.9361,C -1.8466,E1 24.8409,E2 276.8955} C_DIS
LIN {X -106.285,Y 10.4821,Z 112,A 170.3578,B 24.9364,C -1.8417,E1 24.8405,E2 275.2931} C_DIS
LIN {X -106.5089,Y 7.8871,Z 112,A 171.7578,B 24.9367,C -1.8372,E1 24.8402,E2 273.8953} C_DIS
LIN {X -106.6716,Y 5.2481,Z 112,A 173.1933,B 24.937,C -1.8333,E1 24.8399,E2 272.4606} C_DIS
LIN {X -106.7678,Y 2.6447,Z 112,A 174.6036,B 24.9373,C -1.8292,E1 24.8399,E2 271.0515} C_DIS
LIN {X -106.8013,Y 0.0013,Z 112,A 176.0518,B 24.9375,C -1.8257,E1 24.8398,E2 269.603} C_DIS
LIN {X -106.7704,Y -2.5175,Z 112,A 177.3901,B 24.9379,C -1.8209,E1 24.8398,E2 268.2682} C_DIS
LIN {X -106.6733,Y -5.2128,Z 112,A 178.8464,B 24.9381,C -1.8165,E1 24.84,E2 266.8134} C_DIS
LIN {X -106.5144,Y -7.812,Z 112,A -179.7476,B 24.9384,C -1.8124,E1 24.8403,E2 265.4088} C_DIS
LIN {X -106.2946,Y -10.3796,Z 112,A -178.3782,B 24.9388,C -1.8075,E1 24.8406,E2 264.0429} C_DIS
LIN {X -105.9991,Y -13.0599,Z 112,A -176.8967,B 24.939,C -1.8041,E1 24.8411,E2 262.5605} C_DIS
LIN {X -105.6615,Y -15.5531,Z 112,A -175.5343,B 24.9392,C -1.8003,E1 24.8417,E2 261.1991} C_DIS
LIN {X -105.2512,Y -18.1224,Z 112,A -174.1284,B 24.9395,C -1.7963,E1 24.8423,E2 259.7944} C_DIS
LIN {X -104.7653,Y -20.749,Z 112,A -172.6866,B 24.9398,C -1.7921,E1 24.8431,E2 258.3541} C_DIS
LIN {X -104.2265,Y -23.305,Z 112,A -171.2786,B 24.9401,C -1.788,E1 24.8439,E2 256.9476} C_DIS
LIN {X -103.6254,Y -25.8465,Z 112,A -169.8712,B 24.9404,C -1.7839,E1 24.8448,E2 255.5417} C_DIS
LIN {X -103.0105,Y -28.1945,Z 112,A -168.5866,B 24.9407,C -1.7793,E1 24.8457,E2 254.2607} C_DIS
LIN {X -102.2269,Y -30.9184,Z 112,A -167.0235,B 24.9409,C -1.7762,E1 24.847,E2 252.6959} C_DIS
LIN {X -101.4387,Y -33.4137,Z 112,A -165.6131,B 24.9411,C -1.7722,E1 24.8482,E2 251.287} C_DIS
LIN {X -100.5598,Y -35.9739,Z 112,A -164.1539,B 24.9414,C -1.7681,E1 24.8495,E2 249.8291} C_DIS
LIN {X -99.2644,Y -39.4042,Z 112,A -162.1546,B 24.9417,C -1.7636,E1 24.8515,E2 247.8295} C_DIS
LIN {X -98.1606,Y -42.0819,Z 112,A -160.6098,B 24.942,C -1.7587,E1 24.8532,E2 246.2878} C_DIS
LIN {X -97.1034,Y -44.4669,Z 112,A -159.1999,B 24.9423,C -1.7551,E1 24.8548,E2 244.8788} C_DIS
LIN {X -96.0173,Y -46.7649,Z 112,A -157.825,B 24.9425,C -1.7517,E1 24.8565,E2 243.5045} C_DIS
LIN {X -94.8429,Y -49.1029,Z 112,A -156.4156,B 24.9427,C -1.748,E1 24.8583,E2 242.0964} C_DIS
LIN {X -93.6117,Y -51.4114,Z 112,A -155.0105,B 24.943,C -1.7442,E1 24.8601,E2 240.6929} C_DIS
LIN {X -92.4907,Y -53.3993,Z 112,A -153.7182,B 24.943,C -1.7434,E1 24.8619,E2 239.3957} C_DIS
LIN {X -90.9726,Y -55.9487,Z 112,A -152.1704,B 24.9434,C -1.7375,E1 24.8642,E2 237.8539} C_DIS
LIN {X -89.5174,Y -58.2496,Z 112,A -150.7071,B 24.9437,C -1.7338,E1 24.8664,E2 236.3921} C_DIS
LIN {X -88.0648,Y -60.4234,Z 112,A -149.2932,B 24.9439,C -1.7307,E1 24.8686,E2 234.9787} C_DIS
LIN {X -85.787,Y -63.6158,Z 112,A -147.1762,B 24.9442,C -1.7259,E1 24.8721,E2 232.8627} C_DIS
LIN {X -84.1765,Y -65.7317,Z 112,A -145.5527,B 24.9439,C -1.7299,E1 24.8749,E2 231.222} C_DIS
LIN {X -82.083,Y -68.3254,Z 112,A -143.9716,B 24.9447,C -1.7179,E1 24.8776,E2 229.6622} C_DIS
LIN {X -80.0868,Y -70.6566,Z 112,A -142.0942,B 24.9444,C -1.7228,E1 24.8811,E2 227.7645} C_DIS
LIN {X -77.424,Y -73.5648,Z 112,A -140.1601,B 24.9451,C -1.7112,E1 24.8848,E2 225.8496} C_DIS
LIN {X -75.5534,Y -75.4852,Z 112,A -138.7185,B 24.9453,C -1.7083,E1 24.8876,E2 224.4089} C_DIS
LIN {X -73.6163,Y -77.3756,Z 112,A -137.0719,B 24.945,C -1.7127,E1 24.8909,E2 222.745} C_DIS
LIN {X -71.2057,Y -79.5972,Z 112,A -135.4113,B 24.9455,C -1.7054,E1 24.8943,E2 221.095} C_DIS
LIN {X -68.2487,Y -82.1467,Z 112,A -133.4027,B 24.946,C -1.6981,E1 24.8986,E2 219.096} C_DIS
LIN {X -66.2177,Y -83.7925,Z 112,A -131.9726,B 24.946,C -1.6966,E1 24.9017,E2 217.6642} C_DIS
LIN {X -63.697,Y -85.7262,Z 112,A -130.2715,B 24.9463,C -1.6934,E1 24.9055,E2 215.9646} C_DIS
LIN {X -61.5813,Y -87.2583,Z 112,A -128.8651,B 24.9464,C -1.6912,E1 24.9087,E2 214.5585} C_DIS
LIN {X -59.4296,Y -88.7377,Z 112,A -127.4839,B 24.9466,C -1.6882,E1 24.9119,E2 213.1799} C_DIS
LIN {X -56.0303,Y -90.923,Z 112,A -125.2836,B 24.9467,C -1.6861,E1 24.9171,E2 210.9776} C_DIS
LIN {X -54.0062,Y -92.1382,Z 112,A -123.9973,B 24.9467,C -1.685,E1 24.9202,E2 209.6899} C_DIS
LIN {X -51.5747,Y -93.5218,Z 112,A -122.505,B 24.9469,C -1.6826,E1 24.9238,E2 208.1991} C_DIS
LIN {X -49.1908,Y -94.7979,Z 112,A -121.0528,B 24.9471,C -1.6807,E1 24.9274,E2 206.7472} C_DIS
LIN {X -46.9367,Y -95.9334,Z 112,A -119.723,B 24.9472,C -1.6781,E1 24.9307,E2 205.4201} C_DIS
LIN {X -44.476,Y -97.0993,Z 112,A -118.2307,B 24.9472,C -1.6776,E1 24.9345,E2 203.9252} C_DIS
LIN {X -42.4927,Y -97.9815,Z 112,A -117.0163,B 24.9472,C -1.6784,E1 24.9376,E2 202.7061} C_DIS
LIN {X -39.6641,Y -99.1622,Z 112,A -115.4156,B 24.9474,C -1.675,E1 24.9417,E2 201.11} C_DIS
LIN {X -37.2918,Y -100.078,Z 112,A -114.0485,B 24.9474,C -1.6738,E1 24.9453,E2 199.7428} C_DIS
LIN {X -34.8299,Y -100.9612,Z 112,A -112.6401,B 24.9476,C -1.6728,E1 24.949,E2 198.334} C_DIS
LIN {X -32.2615,Y -101.8115,Z 112,A -111.1889,B 24.9476,C -1.6717,E1 24.9529,E2 196.8829} C_DIS
LIN {X -30.0474,Y -102.4853,Z 112,A -109.9159,B 24.9476,C -1.6721,E1 24.9563,E2 195.6068} C_DIS
LIN {X -27.2333,Y -103.2701,Z 112,A -108.3762,B 24.9477,C -1.67,E1 24.9604,E2 194.0698} C_DIS
LIN {X -24.8584,Y -103.8665,Z 112,A -107.0475,B 24.9477,C -1.6699,E1 24.964,E2 192.7394} C_DIS
LIN {X -22.1175,Y -104.4854,Z 112,A -105.5525,B 24.9478,C -1.6686,E1 24.9681,E2 191.2455} C_DIS
LIN {X -19.5509,Y -104.996,Z 112,A -104.1464,B 24.9478,C -1.6682,E1 24.972,E2 189.8389} C_DIS
LIN {X -16.9727,Y -105.4434,Z 112,A -102.7417,B 24.9478,C -1.6678,E1 24.9758,E2 188.4338} C_DIS
LIN {X -13.9556,Y -105.8832,Z 112,A -101.0203,B 24.9477,C -1.6709,E1 24.9806,E2 186.7036} C_DIS
LIN {X -10.4672,Y -106.2865,Z 112,A -99.2211,B 24.9479,C -1.6673,E1 24.9856,E2 184.9121} C_DIS
LIN {X -7.86,Y -106.5111,Z 112,A -97.8168,B 24.9479,C -1.6673,E1 24.9895,E2 183.5072} C_DIS
LIN {X -5.2482,Y -106.6716,Z 112,A -96.2166,B 24.9474,C -1.6753,E1 24.994,E2 181.8875} C_DIS
LIN {X -1.8323,Y -106.7831,Z 112,A -94.5163,B 24.9477,C -1.6702,E1 24.9988,E2 180.1991} C_DIS
LIN {X 0.7511,Y -106.7957,Z 112,A -93.601,B 24.9489,C -1.6514,E1 25.0012,E2 179.3283} C_DIS
Enddeposition()
LIN {X 0.7926,Y -113.0921,Z 113,A -93.1685,B 24.954,C -1.5666,E1 25.0018,E2 179.0968} C_DIS
Startdeposition()
$VEL.CP = VEL_PRINT
LIN {X -0.8773,Y -113.0942,Z 113,A -94.5221,B 24.9553,C -1.5445,E1 24.9979,E2 180.5029} C_DIS
LIN {X -3.6525,Y -113.0386,Z 113,A -95.9279,B 24.9553,C -1.5443,E1 24.994,E2 181.9093} C_DIS
LIN {X -7.8107,Y -112.8276,Z 113,A -97.9739,B 24.9552,C -1.5469,E1 24.9883,E2 183.9497} C_DIS
LIN {X -11.0857,Y -112.555,Z 113,A -99.639,B 24.9552,C -1.5469,E1 24.9837,E2 185.6155} C_DIS
LIN {X -13.8446,Y -112.249,Z 113,A -101.0456,B 24.9552,C -1.5471,E1 24.9798,E2 187.0226} C_DIS
LIN {X -16.0896,Y -111.9473,Z 113,A -102.2571,B 24.9552,C -1.5447,E1 24.9764,E2 188.2408} C_DIS
LIN {X -18.8321,Y -111.5187,Z 113,A -103.6642,B 24.9552,C -1.5451,E1 24.9725,E2 189.6483} C_DIS
LIN {X -21.864,Y -110.9651,Z 113,A -105.1756,B 24.9552,C -1.5478,E1 24.9684,E2 191.155} C_DIS
LIN {X -24.2814,Y -110.4603,Z 113,A -106.4792,B 24.9552,C -1.5461,E1 24.9648,E2 192.464} C_DIS
LIN {X -27.481,Y -109.7102,Z 113,A -108.0828,B 24.955,C -1.5496,E1 24.9605,E2 194.0617} C_DIS
LIN {X -29.6721,Y -109.1359,Z 113,A -109.2952,B 24.9551,C -1.5476,E1 24.9572,E2 195.2807} C_DIS
LIN {X -32.8311,Y -108.2296,Z 113,A -110.8994,B 24.9549,C -1.5513,E1 24.9529,E2 196.8788} C_DIS
LIN {X -36.3086,Y -107.111,Z 113,A -112.8166,B 24.9549,C -1.55,E1 24.9478,E2 198.8025} C_DIS
LIN {X -39.406,Y -106.0127,Z 113,A -114.4215,B 24.9548,C -1.5539,E1 24.9436,E2 200.4013} C_DIS
LIN {X -43.2813,Y -104.4904,Z 113,A -116.5348,B 24.9546,C -1.5559,E1 24.9381,E2 202.5147} C_DIS
LIN {X -46.9189,Y -102.9072,Z 113,A -118.5233,B 24.9545,C -1.559,E1 24.933,E2 204.5005} C_DIS
LIN {X -49.6073,Y -101.6397,Z 113,A -120.0592,B 24.9545,C -1.5595,E1 24.9292,E2 206.0391} C_DIS
LIN {X -52.863,Y -99.9829,Z 113,A -121.9152,B 24.9543,C -1.5617,E1 24.9246,E2 207.8949} C_DIS
LIN {X -55.3008,Y -98.6555,Z 113,A -123.3891,B 24.9543,C -1.5608,E1 24.9209,E2 209.3751} C_DIS
LIN {X -58.1448,Y -97.0088,Z 113,A -124.9957,B 24.9541,C -1.5656,E1 24.9171,E2 210.9752} C_DIS
LIN {X -60.508,Y -95.5526,Z 113,A -126.4067,B 24.954,C -1.5676,E1 24.9137,E2 212.386} C_DIS
LIN {X -62.8348,Y -94.0389,Z 113,A -127.8176,B 24.9538,C -1.5696,E1 24.9105,E2 213.7966} C_DIS
LIN {X -65.8378,Y -91.959,Z 113,A -129.6751,B 24.9537,C -1.5725,E1 24.9062,E2 215.6538} C_DIS
LIN {X -68.0748,Y -90.3155,Z 113,A -131.0868,B 24.9535,C -1.5747,E1 24.903,E2 217.0651} C_DIS
LIN {X -70.6714,Y -88.3011,Z 113,A -132.7583,B 24.9534,C -1.5774,E1 24.8994,E2 218.7363} C_DIS
LIN {X -72.7131,Y -86.6265,Z 113,A -134.107,B 24.9533,C -1.5796,E1 24.8965,E2 220.0851} C_DIS
LIN {X -75.4912,Y -84.2147,Z 113,A -135.9941,B 24.9531,C -1.5823,E1 24.8925,E2 221.9731} C_DIS
LIN {X -77.6148,Y -82.2619,Z 113,A -137.4413,B 24.9529,C -1.5859,E1 24.8896,E2 223.4177} C_DIS
LIN {X -79.9735,Y -79.9735,Z 113,A -139.1137,B 24.9527,C -1.5891,E1 24.8862,E2 225.0895} C_DIS
LIN {X -81.9121,Y -77.9868,Z 113,A -140.5267,B 24.9525,C -1.5918,E1 24.8835,E2 226.502} C_DIS
LIN {X -83.8013,Y -75.9531,Z 113,A -141.9399,B 24.9523,C -1.5947,E1 24.8808,E2 227.9146} C_DIS
LIN {X -85.64,Y -73.8736,Z 113,A -143.3533,B 24.9522,C -1.5977,E1 24.8782,E2 229.3274} C_DIS
LIN {X -87.9796,Y -71.0681,Z 113,A -145.2134,B 24.9519,C -1.6017,E1 24.8749,E2 231.1865} C_DIS
LIN {X -90.0088,Y -68.4831,Z 113,A -146.8868,B 24.9517,C -1.6053,E1 24.8721,E2 232.8592} C_DIS
Enddeposition()
END
